			zyl_rafo_vorschub.fb.st_config.b_aktiv := NOT gst_datensatz.st_md.b_wt_transport_simulation;
			zyl_rafo_vorschub.fb(
				st_config:= ,
				bw_nocken_zylinder_einfahren:= ,
				bw_nocken_zylinder_ausfahren:= ,
				uw_nocken_zylinder_einfahren:= ,
				uw_nocken_zylinder_ausfahren:= ,
				b_direkttaste_ausfahren:= ,
				b_direkttaste_mittefahren:= ,
				b_direkttaste_einfahren	:= ,
				e_druckwaechter:= ST_Betriebsfreigaben.e_druckwaechter,
				i16_betriebsart:= gi16_betriebsart,
				b_no_gesteuert_im_norm_betrieb:= ,
				st_ctrl_in:= zyl_rafo_vorschub.st_ctrl.in,
				b_masterachse_hand_dialog_aktiv:= ,
				st_visu:= visu.st_zyl,
				st_ctrl_out=> zyl_rafo_vorschub.st_ctrl.out,
				a_ventil_einfahren=> a_zyl_vorschub_einfahren,
				a_ventil_ausfahren=> a_zyl_vorschub_ausfahren);
	
			zyl_rafo_kamm.fb.st_config.b_aktiv := NOT gst_datensatz.st_md.b_wt_transport_simulation;
			zyl_rafo_kamm.fb(
				st_config:= ,
				bw_nocken_zylinder_einfahren:= ,
				bw_nocken_zylinder_ausfahren:= ,
				uw_nocken_zylinder_einfahren:= ,
				uw_nocken_zylinder_ausfahren:= ,
				b_direkttaste_ausfahren:= ,
				b_direkttaste_mittefahren:= ,
				b_direkttaste_einfahren	:= ,
				e_druckwaechter:= ST_Betriebsfreigaben.e_druckwaechter,
				i16_betriebsart:= gi16_betriebsart,
				b_no_gesteuert_im_norm_betrieb:= ,
				st_ctrl_in:= zyl_rafo_kamm.st_ctrl.in,
				b_masterachse_hand_dialog_aktiv:= ,
				st_visu:= visu.st_zyl,
				st_ctrl_out=> zyl_rafo_kamm.st_ctrl.out,
				a_ventil_einfahren=> ,
				a_ventil_ausfahren=> );
	
			zyl_rafo_vorzentrierer.fb.st_config.b_aktiv := NOT gst_datensatz.st_md.b_wt_transport_simulation;
			zyl_rafo_vorzentrierer.fb(
				st_config:= ,
				bw_nocken_zylinder_einfahren:= ,
				bw_nocken_zylinder_ausfahren:= ,
				uw_nocken_zylinder_einfahren:= ,
				uw_nocken_zylinder_ausfahren:= ,
				b_direkttaste_ausfahren:= ,
				b_direkttaste_mittefahren:= ,
				b_direkttaste_einfahren	:= ,
				e_druckwaechter:= ST_Betriebsfreigaben.e_druckwaechter,
				i16_betriebsart:= gi16_betriebsart,
				b_no_gesteuert_im_norm_betrieb:= ,
				st_ctrl_in:= zyl_rafo_vorzentrierer.st_ctrl.in,
				b_masterachse_hand_dialog_aktiv:= ,
				st_visu:= visu.st_zyl,
				st_ctrl_out=> zyl_rafo_vorzentrierer.st_ctrl.out,
				a_ventil_einfahren=> ,
				a_ventil_ausfahren=> );
	END_CASE
END_IF
END_PROGRAM

(* POU Gemeinsamkeiten17xx/Initialisierung/Startup/ST_Datainit_Zylinder, ST *)
PROGRAM ST_Datainit_Zylinder
VAR
	b_config_fertig			: BOOL := FALSE;
END_VAR
IF	NOT zyl_wt_zentrierer_tisch.fb.st_config.b_config_fertig OR
	NOT zyl_wt_stopper_tisch.fb.st_config.b_config_fertig OR
	NOT zyl_wt_stopper_auslauf.fb.st_config.b_config_fertig OR
	NOT zyl_hublift_rechts_lift.fb.st_config.b_config_fertig OR
	NOT zyl_hublift_rechts_wt_einzug.fb.st_config.b_config_fertig OR
	NOT zyl_hublift_rechts_wt_klinke.fb.st_config.b_config_fertig OR
	NOT zyl_hublift_links_lift.fb.st_config.b_config_fertig OR
	NOT zyl_hublift_links_wt_einzug.fb.st_config.b_config_fertig OR
	NOT zyl_hublift_links_wt_klinke.fb.st_config.b_config_fertig OR
	NOT zyl_hublift_links_stopper.fb.st_config.b_config_fertig OR
	NOT zyl_hublift_links_eingriffschutz.fb.st_config.b_config_fertig OR
	NOT zyl_haspel_li_heben.fb.st_config.b_config_fertig OR
	NOT zyl_haspel_li_abspulen.fb.st_config.b_config_fertig OR
	NOT zyl_haspel_li_sperren.fb.st_config.b_config_fertig OR
	NOT zyl_haspel_re_heben.fb.st_config.b_config_fertig OR
	NOT zyl_haspel_re_abspulen.fb.st_config.b_config_fertig OR
	NOT zyl_haspel_re_sperren.fb.st_config.b_config_fertig OR
	NOT zyl_haspel_verschieben.fb.st_config.b_config_fertig OR
	NOT zyl_bandeinzuege_verschieben.fb.st_config.b_config_fertig OR
	NOT zyl_bawe_vorschub.fb.st_config.b_config_fertig OR
	NOT zyl_bawe_querschub.fb.st_config.b_config_fertig OR
	NOT zyl_bawe_faenger_li.fb.st_config.b_config_fertig OR
	NOT zyl_bawe_faenger_re.fb.st_config.b_config_fertig OR
	NOT zyl_bawe_halter_li.fb.st_config.b_config_fertig OR
	NOT zyl_bawe_halter_re.fb.st_config.b_config_fertig OR
	NOT zyl_wt_stopper_einlauf.fb.st_config.b_config_fertig OR
	NOT zyl_rafo_faenger.fb.st_config.b_config_fertig OR
	NOT zyl_rafo_klemmen.fb.st_config.b_config_fertig OR
	NOT zyl_rafo_vorschub.fb.st_config.b_config_fertig OR
	NOT zyl_rafo_kamm.fb.st_config.b_config_fertig OR
	NOT zyl_rafo_vorzentrierer.fb.st_config.b_config_fertig OR
	NOT zyl_Indexier_Bestueckpos.fb.st_config.b_config_fertig OR
	NOT zyl_Indexier_Einlauf.fb.st_config.b_config_fertig
	THEN

		(* WT Zentrierzylinder am Tisch *)
		zyl_wt_zentrierer_tisch.fb.st_config.b_config_fertig := FALSE;
		zyl_wt_zentrierer_tisch.fb.st_config.b_endlage1_aktiv := FALSE;
		zyl_wt_zentrierer_tisch.fb.st_config.b_endlage2_aktiv := FALSE;
		zyl_wt_zentrierer_tisch.fb.st_config.b_sensor1_aktiv := TRUE;
		zyl_wt_zentrierer_tisch.fb.st_config.b_sensor2_aktiv := TRUE;
		zyl_wt_zentrierer_tisch.fb.st_config.i16_gruppe := 3;
		zyl_wt_zentrierer_tisch.fb.st_config.i16_identnummer := 15;
		zyl_wt_zentrierer_tisch.fb.st_config.i16_meld_startindex := 2280;
		zyl_wt_zentrierer_tisch.fb.st_config.str_beschreibung := ' ';
		zyl_wt_zentrierer_tisch.fb.st_config.str_instanz_name := 'WT Zentrierzylinder am Tisch';
		zyl_wt_zentrierer_tisch.fb.st_config.str_zylinder_typ := '2V4E_EIN_AUS';
		zyl_wt_zentrierer_tisch.fb.st_config.t_ein_aus_fahrzeit := t#0ms;
		zyl_wt_zentrierer_tisch.fb.st_config.t_ueberwachungszeit := t#1000ms;
		zyl_wt_zentrierer_tisch.fb.st_config.i16_tzk_faktor_ausfahren := 100;
		zyl_wt_zentrierer_tisch.fb.st_config.i16_tzk_faktor_einfahren := 100;
		zyl_wt_zentrierer_tisch.fb.st_config.b_config_fertig := TRUE;
		
		(* WT Stoppzylinder am Tisch *)
		zyl_wt_stopper_tisch.fb.st_config.b_config_fertig := FALSE;
		zyl_wt_stopper_tisch.fb.st_config.b_endlage1_aktiv := FALSE;
		zyl_wt_stopper_tisch.fb.st_config.b_endlage2_aktiv := FALSE;
		zyl_wt_stopper_tisch.fb.st_config.b_sensor1_aktiv := TRUE;
		zyl_wt_stopper_tisch.fb.st_config.b_sensor2_aktiv := FALSE;
		zyl_wt_stopper_tisch.fb.st_config.i16_gruppe := 3;
		zyl_wt_stopper_tisch.fb.st_config.i16_identnummer := 16;
		zyl_wt_stopper_tisch.fb.st_config.i16_meld_startindex := 2300;
		zyl_wt_stopper_tisch.fb.st_config.str_beschreibung := ' ';
		zyl_wt_stopper_tisch.fb.st_config.str_instanz_name := 'WT Stoppzylinder am Tisch';

		zyl_wt_stopper_tisch.fb.st_config.t_ein_aus_fahrzeit := t#0ms;
		zyl_wt_stopper_tisch.fb.st_config.t_ueberwachungszeit := t#1000ms;
		zyl_wt_stopper_tisch.fb.st_config.i16_tzk_faktor_ausfahren := 100;
		zyl_wt_stopper_tisch.fb.st_config.i16_tzk_faktor_einfahren := 100;


		IF gst_Datensatz.st_md.b_anwahl_transport_achse THEN
			zyl_wt_stopper_tisch.fb.st_config.str_zylinder_typ := '1V0E_NO';
		ELSE
			zyl_wt_stopper_tisch.fb.st_config.str_zylinder_typ := '2V2E_EIN_AUS';
		END_IF

		zyl_wt_stopper_tisch.fb.st_config.b_config_fertig := TRUE;

		(* WT Stopperzylinder am Auslauf *)
		CASE gst_datensatz.st_md.i16_typ_zelle OF
			KEINE_ZELLE:
				;
			BESTUECKZELLE_1700, RASTERFOLIE:
				zyl_wt_stopper_auslauf.fb.st_config.b_config_fertig := FALSE;
				zyl_wt_stopper_auslauf.fb.st_config.b_endlage1_aktiv := FALSE;
				zyl_wt_stopper_auslauf.fb.st_config.b_endlage2_aktiv := FALSE;
				zyl_wt_stopper_auslauf.fb.st_config.b_sensor1_aktiv := FALSE;
				zyl_wt_stopper_auslauf.fb.st_config.b_sensor2_aktiv := FALSE;
				zyl_wt_stopper_auslauf.fb.st_config.i16_gruppe := 3;
				zyl_wt_stopper_auslauf.fb.st_config.i16_identnummer := 17;
				zyl_wt_stopper_auslauf.fb.st_config.i16_meld_startindex := 2320;
				zyl_wt_stopper_auslauf.fb.st_config.str_beschreibung := ' ';
				zyl_wt_stopper_auslauf.fb.st_config.str_instanz_name := 'WT Stopperzylinder am Auslauf';
				zyl_wt_stopper_auslauf.fb.st_config.str_zylinder_typ := '2V0E';
				zyl_wt_stopper_auslauf.fb.st_config.t_ein_aus_fahrzeit := t#150ms;
				zyl_wt_stopper_auslauf.fb.st_config.t_ueberwachungszeit := t#1000ms;
				zyl_wt_stopper_auslauf.fb.st_config.i16_tzk_faktor_ausfahren := 100;
				zyl_wt_stopper_auslauf.fb.st_config.i16_tzk_faktor_einfahren := 100;
				zyl_wt_stopper_auslauf.fb.st_config.b_config_fertig := TRUE;

			BESTUECKZELLE_1720:
				zyl_wt_stopper_auslauf.fb.st_config.b_config_fertig := FALSE;
				zyl_wt_stopper_auslauf.fb.st_config.b_endlage1_aktiv := FALSE;
				zyl_wt_stopper_auslauf.fb.st_config.b_endlage2_aktiv := FALSE;
				zyl_wt_stopper_auslauf.fb.st_config.b_sensor1_aktiv := FALSE;
				zyl_wt_stopper_auslauf.fb.st_config.b_sensor2_aktiv := FALSE;
				zyl_wt_stopper_auslauf.fb.st_config.i16_gruppe := 3;
				zyl_wt_stopper_auslauf.fb.st_config.i16_identnummer := 17;
				zyl_wt_stopper_auslauf.fb.st_config.i16_meld_startindex := 2320;
				zyl_wt_stopper_auslauf.fb.st_config.str_beschreibung := ' ';
				zyl_wt_stopper_auslauf.fb.st_config.str_instanz_name := 'WT Stopperzylinder am Auslauf';
				zyl_wt_stopper_auslauf.fb.st_config.str_zylinder_typ := '2V2E_EIN_AUS';
				zyl_wt_stopper_auslauf.fb.st_config.t_ein_aus_fahrzeit := t#150ms;
				zyl_wt_stopper_auslauf.fb.st_config.t_ueberwachungszeit := t#1000ms;
				zyl_wt_stopper_auslauf.fb.st_config.i16_tzk_faktor_ausfahren := 100;
				zyl_wt_stopper_auslauf.fb.st_config.i16_tzk_faktor_einfahren := 100;
				zyl_wt_stopper_auslauf.fb.st_config.b_config_fertig := TRUE;
		END_CASE

		(* Hublift-Lift rechts *)
		zyl_hublift_rechts_lift.fb.st_config.b_config_fertig := FALSE;
		zyl_hublift_rechts_lift.fb.st_config.b_endlage1_aktiv := TRUE;
		zyl_hublift_rechts_lift.fb.st_config.b_endlage2_aktiv := FALSE;
		zyl_hublift_rechts_lift.fb.st_config.b_sensor1_aktiv := TRUE;
		zyl_hublift_rechts_lift.fb.st_config.b_sensor2_aktiv := FALSE;
		zyl_hublift_rechts_lift.fb.st_config.i16_gruppe := 4;
		zyl_hublift_rechts_lift.fb.st_config.i16_identnummer := 18;
		zyl_hublift_rechts_lift.fb.st_config.i16_meld_startindex := 2340;
		zyl_hublift_rechts_lift.fb.st_config.str_beschreibung := ' ';
		zyl_hublift_rechts_lift.fb.st_config.str_instanz_name := 'Hublift-Lift rechts';
		zyl_hublift_rechts_lift.fb.st_config.str_zylinder_typ := '2V2E_EIN_AUS';
		zyl_hublift_rechts_lift.fb.st_config.t_ein_aus_fahrzeit := t#0ms;
		zyl_hublift_rechts_lift.fb.st_config.t_ueberwachungszeit := t#3500ms;
		zyl_hublift_rechts_lift.fb.st_config.i16_tzk_faktor_ausfahren := 100;
		zyl_hublift_rechts_lift.fb.st_config.i16_tzk_faktor_einfahren := 100;
		zyl_hublift_rechts_lift.fb.st_config.b_config_fertig := TRUE;
		
		(* Hublift-WT-Einzug rechts *)
		zyl_hublift_rechts_wt_einzug.fb.st_config.b_config_fertig := FALSE;
		zyl_hublift_rechts_wt_einzug.fb.st_config.b_endlage1_aktiv := TRUE;
		zyl_hublift_rechts_wt_einzug.fb.st_config.b_endlage2_aktiv := FALSE;
		zyl_hublift_rechts_wt_einzug.fb.st_config.b_sensor1_aktiv := TRUE;
		zyl_hublift_rechts_wt_einzug.fb.st_config.b_sensor2_aktiv := FALSE;
		zyl_hublift_rechts_wt_einzug.fb.st_config.i16_gruppe := 4;
		zyl_hublift_rechts_wt_einzug.fb.st_config.i16_identnummer := 19;
		zyl_hublift_rechts_wt_einzug.fb.st_config.i16_meld_startindex := 2360;
		zyl_hublift_rechts_wt_einzug.fb.st_config.str_beschreibung := ' ';
		zyl_hublift_rechts_wt_einzug.fb.st_config.str_instanz_name := 'Hublift-WT-Einzug rechts';
		zyl_hublift_rechts_wt_einzug.fb.st_config.str_zylinder_typ := '2V2E_EIN_AUS';
		zyl_hublift_rechts_wt_einzug.fb.st_config.t_ein_aus_fahrzeit := t#0ms;
		zyl_hublift_rechts_wt_einzug.fb.st_config.t_ueberwachungszeit := t#2500ms;
		zyl_hublift_rechts_wt_einzug.fb.st_config.i16_tzk_faktor_ausfahren := 100;
		zyl_hublift_rechts_wt_einzug.fb.st_config.i16_tzk_faktor_einfahren := 100;
		zyl_hublift_rechts_wt_einzug.fb.st_config.b_config_fertig := TRUE;
		
		(* Hublift-WT-Klinke rechts *)
		zyl_hublift_rechts_wt_klinke.fb.st_config.b_config_fertig := FALSE;
		zyl_hublift_rechts_wt_klinke.fb.st_config.b_endlage1_aktiv := TRUE;
		zyl_hublift_rechts_wt_klinke.fb.st_config.b_endlage2_aktiv := FALSE;
		zyl_hublift_rechts_wt_klinke.fb.st_config.b_sensor1_aktiv := TRUE;
		zyl_hublift_rechts_wt_klinke.fb.st_config.b_sensor2_aktiv := FALSE;
		zyl_hublift_rechts_wt_klinke.fb.st_config.i16_gruppe := 4;
		zyl_hublift_rechts_wt_klinke.fb.st_config.i16_identnummer := 20;
		zyl_hublift_rechts_wt_klinke.fb.st_config.i16_meld_startindex := 2380;
		zyl_hublift_rechts_wt_klinke.fb.st_config.str_beschreibung := ' ';
		zyl_hublift_rechts_wt_klinke.fb.st_config.str_instanz_name := 'Hublift-WT-Klinke rechts';
		zyl_hublift_rechts_wt_klinke.fb.st_config.str_zylinder_typ := '2V2E_EIN_AUS';
		zyl_hublift_rechts_wt_klinke.fb.st_config.t_ein_aus_fahrzeit := t#0ms;
		zyl_hublift_rechts_wt_klinke.fb.st_config.t_ueberwachungszeit := t#1500ms;
		zyl_hublift_rechts_wt_klinke.fb.st_config.i16_tzk_faktor_ausfahren := 100;
		zyl_hublift_rechts_wt_klinke.fb.st_config.i16_tzk_faktor_einfahren := 100;
		zyl_hublift_rechts_wt_klinke.fb.st_config.b_config_fertig := TRUE;
		
		(* Hublift-Lift links *)
		zyl_hublift_links_lift.fb.st_config.b_config_fertig := FALSE;
		zyl_hublift_links_lift.fb.st_config.b_endlage1_aktiv := TRUE;
		zyl_hublift_links_lift.fb.st_config.b_endlage2_aktiv := FALSE;
		zyl_hublift_links_lift.fb.st_config.b_sensor1_aktiv := TRUE;
		zyl_hublift_links_lift.fb.st_config.b_sensor2_aktiv := FALSE;
		zyl_hublift_links_lift.fb.st_config.i16_gruppe := 4;
		zyl_hublift_links_lift.fb.st_config.i16_identnummer := 21;
		zyl_hublift_links_lift.fb.st_config.i16_meld_startindex := 2400;
		zyl_hublift_links_lift.fb.st_config.str_beschreibung := ' ';
		zyl_hublift_links_lift.fb.st_config.str_instanz_name := 'Hublift-Lift links';
		zyl_hublift_links_lift.fb.st_config.str_zylinder_typ := '2V2E_EIN_AUS';
		zyl_hublift_links_lift.fb.st_config.t_ein_aus_fahrzeit := t#0ms;
		zyl_hublift_links_lift.fb.st_config.t_ueberwachungszeit := t#3500ms;
		zyl_hublift_links_lift.fb.st_config.i16_tzk_faktor_ausfahren := 100;
		zyl_hublift_links_lift.fb.st_config.i16_tzk_faktor_einfahren := 100;
		zyl_hublift_links_lift.fb.st_config.b_config_fertig := TRUE;
		
		(* Hublift-WT-Einzug links *)
		zyl_hublift_links_wt_einzug.fb.st_config.b_config_fertig := FALSE;
		zyl_hublift_links_wt_einzug.fb.st_config.b_endlage1_aktiv := TRUE;
		zyl_hublift_links_wt_einzug.fb.st_config.b_endlage2_aktiv := FALSE;
		zyl_hublift_links_wt_einzug.fb.st_config.b_sensor1_aktiv := TRUE;
		zyl_hublift_links_wt_einzug.fb.st_config.b_sensor2_aktiv := FALSE;
		zyl_hublift_links_wt_einzug.fb.st_config.i16_gruppe := 4;
		zyl_hublift_links_wt_einzug.fb.st_config.i16_identnummer := 22;
		zyl_hublift_links_wt_einzug.fb.st_config.i16_meld_startindex := 2420;
		zyl_hublift_links_wt_einzug.fb.st_config.str_beschreibung := ' ';
		zyl_hublift_links_wt_einzug.fb.st_config.str_instanz_name := 'Hublift-WT-Einzug links';
		zyl_hublift_links_wt_einzug.fb.st_config.str_zylinder_typ := '2V2E_EIN_AUS';
		zyl_hublift_links_wt_einzug.fb.st_config.t_ein_aus_fahrzeit := t#0ms;
		zyl_hublift_links_wt_einzug.fb.st_config.t_ueberwachungszeit := t#2500ms;
		zyl_hublift_links_wt_einzug.fb.st_config.i16_tzk_faktor_ausfahren := 100;
		zyl_hublift_links_wt_einzug.fb.st_config.i16_tzk_faktor_einfahren := 100;
		zyl_hublift_links_wt_einzug.fb.st_config.b_config_fertig := TRUE;

		(* Hublift-WT-Klinke links *)
		zyl_hublift_links_wt_klinke.fb.st_config.b_config_fertig := FALSE;
		zyl_hublift_links_wt_klinke.fb.st_config.b_endlage1_aktiv := TRUE;
		zyl_hublift_links_wt_klinke.fb.st_config.b_endlage2_aktiv := FALSE;
		zyl_hublift_links_wt_klinke.fb.st_config.b_sensor1_aktiv := TRUE;
		zyl_hublift_links_wt_klinke.fb.st_config.b_sensor2_aktiv := FALSE;
		zyl_hublift_links_wt_klinke.fb.st_config.i16_gruppe := 4;
		zyl_hublift_links_wt_klinke.fb.st_config.i16_identnummer := 23;
		zyl_hublift_links_wt_klinke.fb.st_config.i16_meld_startindex := 2440;
		zyl_hublift_links_wt_klinke.fb.st_config.str_beschreibung := ' ';
		zyl_hublift_links_wt_klinke.fb.st_config.str_instanz_name := 'Hublift-WT-Klinke links';
		zyl_hublift_links_wt_klinke.fb.st_config.str_zylinder_typ := '2V2E_EIN_AUS';
		zyl_hublift_links_wt_klinke.fb.st_config.t_ein_aus_fahrzeit := t#0ms;
		zyl_hublift_links_wt_klinke.fb.st_config.t_ueberwachungszeit := t#1500ms;
		zyl_hublift_links_wt_klinke.fb.st_config.i16_tzk_faktor_ausfahren := 100;
		zyl_hublift_links_wt_klinke.fb.st_config.i16_tzk_faktor_einfahren := 100;
		zyl_hublift_links_wt_klinke.fb.st_config.b_config_fertig := TRUE;

		(* Hublift-Stopper links *)
		zyl_hublift_links_stopper.fb.st_config.b_config_fertig := FALSE;
		zyl_hublift_links_stopper.fb.st_config.b_endlage1_aktiv := TRUE;
		zyl_hublift_links_stopper.fb.st_config.b_endlage2_aktiv := FALSE;
		zyl_hublift_links_stopper.fb.st_config.b_sensor1_aktiv := TRUE;
		zyl_hublift_links_stopper.fb.st_config.b_sensor2_aktiv := FALSE;
		zyl_hublift_links_stopper.fb.st_config.i16_gruppe := 4;
		zyl_hublift_links_stopper.fb.st_config.i16_identnummer := 24;
		zyl_hublift_links_stopper.fb.st_config.i16_meld_startindex := 2460;
		zyl_hublift_links_stopper.fb.st_config.str_beschreibung := ' ';
		zyl_hublift_links_stopper.fb.st_config.str_instanz_name := 'Hublift-Stopper links';
		zyl_hublift_links_stopper.fb.st_config.str_zylinder_typ := '2V2E_EIN_AUS';
		zyl_hublift_links_stopper.fb.st_config.t_ein_aus_fahrzeit := t#0ms;
		zyl_hublift_links_stopper.fb.st_config.t_ueberwachungszeit := t#2000ms;
		zyl_hublift_links_stopper.fb.st_config.i16_tzk_faktor_ausfahren := 100;
		zyl_hublift_links_stopper.fb.st_config.i16_tzk_faktor_einfahren := 100;
		zyl_hublift_links_stopper.fb.st_config.b_config_fertig := TRUE;

		(* zyl_hublift_links_eingriffschutz *)
		zyl_hublift_links_eingriffschutz.fb.st_config.b_config_fertig := FALSE;
		zyl_hublift_links_eingriffschutz.fb.st_config.b_endlage1_aktiv := TRUE;
		zyl_hublift_links_eingriffschutz.fb.st_config.b_endlage2_aktiv := FALSE;
		zyl_hublift_links_eingriffschutz.fb.st_config.b_sensor1_aktiv := TRUE;
		zyl_hublift_links_eingriffschutz.fb.st_config.b_sensor2_aktiv := FALSE;
		zyl_hublift_links_eingriffschutz.fb.st_config.i16_gruppe := 4;
		zyl_hublift_links_eingriffschutz.fb.st_config.i16_identnummer := 44;
		zyl_hublift_links_eingriffschutz.fb.st_config.i16_meld_startindex := 2860;
		zyl_hublift_links_eingriffschutz.fb.st_config.str_beschreibung := ' ';
		zyl_hublift_links_eingriffschutz.fb.st_config.str_instanz_name := 'Hublift links Eingriffschutz';
		zyl_hublift_links_eingriffschutz.fb.st_config.str_zylinder_typ := '2V2E_EIN_AUS';
		zyl_hublift_links_eingriffschutz.fb.st_config.t_ein_aus_fahrzeit := t#0ms;
		zyl_hublift_links_eingriffschutz.fb.st_config.t_ueberwachungszeit := t#4000ms;
		zyl_hublift_links_eingriffschutz.fb.st_config.i16_tzk_faktor_ausfahren := 100;
		zyl_hublift_links_eingriffschutz.fb.st_config.i16_tzk_faktor_einfahren := 100;
		zyl_hublift_links_eingriffschutz.fb.st_config.b_config_fertig := TRUE;
		
		(* Haspel links heben *)
		zyl_haspel_li_heben.fb.st_config.b_config_fertig := FALSE;
		zyl_haspel_li_heben.fb.st_config.b_endlage1_aktiv := FALSE;
		zyl_haspel_li_heben.fb.st_config.b_endlage2_aktiv := FALSE;
		zyl_haspel_li_heben.fb.st_config.b_sensor1_aktiv := FALSE;
		zyl_haspel_li_heben.fb.st_config.b_sensor2_aktiv := FALSE;
		zyl_haspel_li_heben.fb.st_config.i16_gruppe := 2;
		zyl_haspel_li_heben.fb.st_config.i16_identnummer := 7;
		zyl_haspel_li_heben.fb.st_config.i16_meld_startindex := 2120;
		zyl_haspel_li_heben.fb.st_config.str_beschreibung := ' ';
		zyl_haspel_li_heben.fb.st_config.str_instanz_name := 'Haspel links heben';
		zyl_haspel_li_heben.fb.st_config.str_zylinder_typ := '2V1E_AUS';
		zyl_haspel_li_heben.fb.st_config.t_ein_aus_fahrzeit := t#0ms;
		zyl_haspel_li_heben.fb.st_config.t_ueberwachungszeit := t#8s;
		zyl_haspel_li_heben.fb.st_config.i16_tzk_faktor_ausfahren := 100;
		zyl_haspel_li_heben.fb.st_config.i16_tzk_faktor_einfahren := 100;
		zyl_haspel_li_heben.fb.st_config.b_config_fertig := TRUE;
		
		(* Haspel links abspulen *)
		zyl_haspel_li_abspulen.fb.st_config.b_config_fertig := FALSE;
		zyl_haspel_li_abspulen.fb.st_config.b_endlage1_aktiv := FALSE;
		zyl_haspel_li_abspulen.fb.st_config.b_endlage2_aktiv := FALSE;
		zyl_haspel_li_abspulen.fb.st_config.b_sensor1_aktiv := FALSE;
		zyl_haspel_li_abspulen.fb.st_config.b_sensor2_aktiv := FALSE;
		zyl_haspel_li_abspulen.fb.st_config.i16_gruppe := 2;
		zyl_haspel_li_abspulen.fb.st_config.i16_identnummer := 8;
		zyl_haspel_li_abspulen.fb.st_config.i16_meld_startindex := 2140;
		zyl_haspel_li_abspulen.fb.st_config.str_beschreibung := ' ';
		zyl_haspel_li_abspulen.fb.st_config.str_instanz_name := 'Haspel links abspulen';
		zyl_haspel_li_abspulen.fb.st_config.str_zylinder_typ := '2V1E_AUS';
		zyl_haspel_li_abspulen.fb.st_config.t_ein_aus_fahrzeit := t#0ms;
		zyl_haspel_li_abspulen.fb.st_config.t_ueberwachungszeit := t#3s;
		zyl_haspel_li_abspulen.fb.st_config.i16_tzk_faktor_ausfahren := 100;
		zyl_haspel_li_abspulen.fb.st_config.i16_tzk_faktor_einfahren := 100;
		zyl_haspel_li_abspulen.fb.st_config.b_config_fertig := TRUE;
		
		(* Haspel links sperren *)
		zyl_haspel_li_sperren.fb.st_config.b_config_fertig := FALSE;
		zyl_haspel_li_sperren.fb.st_config.b_endlage1_aktiv := FALSE;
		zyl_haspel_li_sperren.fb.st_config.b_endlage2_aktiv := FALSE;
		zyl_haspel_li_sperren.fb.st_config.b_sensor1_aktiv := TRUE;
		zyl_haspel_li_sperren.fb.st_config.b_sensor2_aktiv := FALSE;
		zyl_haspel_li_sperren.fb.st_config.i16_gruppe := 2;
		zyl_haspel_li_sperren.fb.st_config.i16_identnummer := 9;
		zyl_haspel_li_sperren.fb.st_config.i16_meld_startindex := 2160;
		zyl_haspel_li_sperren.fb.st_config.str_beschreibung := ' ';
		zyl_haspel_li_sperren.fb.st_config.str_instanz_name := 'Haspel links sperren';
		zyl_haspel_li_sperren.fb.st_config.str_zylinder_typ := '2V2E_EIN_AUS';
		zyl_haspel_li_sperren.fb.st_config.t_ein_aus_fahrzeit := t#0ms;
		zyl_haspel_li_sperren.fb.st_config.t_ueberwachungszeit := t#1000ms;
		zyl_haspel_li_sperren.fb.st_config.i16_tzk_faktor_ausfahren := 100;
		zyl_haspel_li_sperren.fb.st_config.i16_tzk_faktor_einfahren := 100;
		zyl_haspel_li_sperren.fb.st_config.b_config_fertig := TRUE;
		
		(* Haspel rechts heben *)
		zyl_haspel_re_heben.fb.st_config.b_config_fertig := FALSE;
		zyl_haspel_re_heben.fb.st_config.b_endlage1_aktiv := FALSE;
		zyl_haspel_re_heben.fb.st_config.b_endlage2_aktiv := FALSE;
		zyl_haspel_re_heben.fb.st_config.b_sensor1_aktiv := FALSE;
		zyl_haspel_re_heben.fb.st_config.b_sensor2_aktiv := FALSE;
		zyl_haspel_re_heben.fb.st_config.i16_gruppe := 2;
		zyl_haspel_re_heben.fb.st_config.i16_identnummer := 10;
		zyl_haspel_re_heben.fb.st_config.i16_meld_startindex := 2180;
		zyl_haspel_re_heben.fb.st_config.str_beschreibung := ' ';
		zyl_haspel_re_heben.fb.st_config.str_instanz_name := 'Haspel rechts heben';
		zyl_haspel_re_heben.fb.st_config.str_zylinder_typ := '2V1E_AUS';
		zyl_haspel_re_heben.fb.st_config.t_ein_aus_fahrzeit := t#0ms;
		zyl_haspel_re_heben.fb.st_config.t_ueberwachungszeit := t#8s;
		zyl_haspel_re_heben.fb.st_config.i16_tzk_faktor_ausfahren := 100;
		zyl_haspel_re_heben.fb.st_config.i16_tzk_faktor_einfahren := 100;
		zyl_haspel_re_heben.fb.st_config.b_config_fertig := TRUE;
		
		(* Haspel rechts abspulen *)
		zyl_haspel_re_abspulen.fb.st_config.b_config_fertig := FALSE;
		zyl_haspel_re_abspulen.fb.st_config.b_endlage1_aktiv := FALSE;
		zyl_haspel_re_abspulen.fb.st_config.b_endlage2_aktiv := FALSE;
		zyl_haspel_re_abspulen.fb.st_config.b_sensor1_aktiv := FALSE;
		zyl_haspel_re_abspulen.fb.st_config.b_sensor2_aktiv := FALSE;
		zyl_haspel_re_abspulen.fb.st_config.i16_gruppe := 2;
		zyl_haspel_re_abspulen.fb.st_config.i16_identnummer := 11;
		zyl_haspel_re_abspulen.fb.st_config.i16_meld_startindex := 2200;
		zyl_haspel_re_abspulen.fb.st_config.str_beschreibung := ' ';
		zyl_haspel_re_abspulen.fb.st_config.str_instanz_name := 'Haspel rechts abspulen';
		zyl_haspel_re_abspulen.fb.st_config.str_zylinder_typ := '2V1E_AUS';
		zyl_haspel_re_abspulen.fb.st_config.t_ein_aus_fahrzeit := t#0ms;
		zyl_haspel_re_abspulen.fb.st_config.t_ueberwachungszeit := t#3s;
		zyl_haspel_re_abspulen.fb.st_config.i16_tzk_faktor_ausfahren := 100;
		zyl_haspel_re_abspulen.fb.st_config.i16_tzk_faktor_einfahren := 100;
		zyl_haspel_re_abspulen.fb.st_config.b_config_fertig := TRUE;
		
		(* Haspel rechts sperren *)
		zyl_haspel_re_sperren.fb.st_config.b_config_fertig := FALSE;
		zyl_haspel_re_sperren.fb.st_config.b_endlage1_aktiv := FALSE;
		zyl_haspel_re_sperren.fb.st_config.b_endlage2_aktiv := FALSE;
		zyl_haspel_re_sperren.fb.st_config.b_sensor1_aktiv := FALSE;
		zyl_haspel_re_sperren.fb.st_config.b_sensor2_aktiv := FALSE;
		zyl_haspel_re_sperren.fb.st_config.i16_gruppe := 2;
		zyl_haspel_re_sperren.fb.st_config.i16_identnummer := 12;
		zyl_haspel_re_sperren.fb.st_config.i16_meld_startindex := 2220;
		zyl_haspel_re_sperren.fb.st_config.str_beschreibung := ' ';
		zyl_haspel_re_sperren.fb.st_config.str_instanz_name := 'Haspel rechts sperren';
		zyl_haspel_re_sperren.fb.st_config.str_zylinder_typ := '2V2E_EIN_AUS';
		zyl_haspel_re_sperren.fb.st_config.t_ein_aus_fahrzeit := t#0ms;
		zyl_haspel_re_sperren.fb.st_config.t_ueberwachungszeit := t#1000ms;
		zyl_haspel_re_sperren.fb.st_config.i16_tzk_faktor_ausfahren := 100;
		zyl_haspel_re_sperren.fb.st_config.i16_tzk_faktor_einfahren := 100;
		zyl_haspel_re_sperren.fb.st_config.b_config_fertig := TRUE;
		
		(* Haspel verschieben *)
		zyl_haspel_verschieben.fb.st_config.b_config_fertig := FALSE;
		zyl_haspel_verschieben.fb.st_config.b_endlage1_aktiv := FALSE;
		zyl_haspel_verschieben.fb.st_config.b_endlage2_aktiv := FALSE;
		zyl_haspel_verschieben.fb.st_config.b_sensor1_aktiv := TRUE;
		zyl_haspel_verschieben.fb.st_config.b_sensor2_aktiv := FALSE;
		zyl_haspel_verschieben.fb.st_config.i16_gruppe := 2;
		zyl_haspel_verschieben.fb.st_config.i16_identnummer := 13;
		zyl_haspel_verschieben.fb.st_config.i16_meld_startindex := 2240;
		zyl_haspel_verschieben.fb.st_config.str_beschreibung := ' ';
		zyl_haspel_verschieben.fb.st_config.str_instanz_name := 'Haspel verschieben';
		zyl_haspel_verschieben.fb.st_config.str_zylinder_typ := '2V2E_EIN_AUS';
		zyl_haspel_verschieben.fb.st_config.t_ein_aus_fahrzeit := t#0ms;
		zyl_haspel_verschieben.fb.st_config.t_ueberwachungszeit := t#8s;
		zyl_haspel_verschieben.fb.st_config.i16_tzk_faktor_ausfahren := 100;
		zyl_haspel_verschieben.fb.st_config.i16_tzk_faktor_einfahren := 100;
		zyl_haspel_verschieben.fb.st_config.b_config_fertig := TRUE;
		
		(* Bandeinzüge verschieben *)
		zyl_bandeinzuege_verschieben.fb.st_config.b_config_fertig := FALSE;
		zyl_bandeinzuege_verschieben.fb.st_config.b_endlage1_aktiv := FALSE;
		zyl_bandeinzuege_verschieben.fb.st_config.b_endlage2_aktiv := FALSE;
		zyl_bandeinzuege_verschieben.fb.st_config.b_sensor1_aktiv := TRUE;
		zyl_bandeinzuege_verschieben.fb.st_config.b_sensor2_aktiv := FALSE;
		zyl_bandeinzuege_verschieben.fb.st_config.i16_gruppe := 2;
		zyl_bandeinzuege_verschieben.fb.st_config.i16_identnummer := 14;
		zyl_bandeinzuege_verschieben.fb.st_config.i16_meld_startindex := 2260;
		zyl_bandeinzuege_verschieben.fb.st_config.str_beschreibung := ' ';
		zyl_bandeinzuege_verschieben.fb.st_config.str_instanz_name := 'Bandeinzüge verschieben';
		zyl_bandeinzuege_verschieben.fb.st_config.str_zylinder_typ := '2V2E_EIN_AUS';
		zyl_bandeinzuege_verschieben.fb.st_config.t_ein_aus_fahrzeit := t#0ms;
		zyl_bandeinzuege_verschieben.fb.st_config.t_ueberwachungszeit := t#8000ms;
		zyl_bandeinzuege_verschieben.fb.st_config.i16_tzk_faktor_ausfahren := 100;
		zyl_bandeinzuege_verschieben.fb.st_config.i16_tzk_faktor_einfahren := 100;
		zyl_bandeinzuege_verschieben.fb.st_config.b_config_fertig := TRUE;
		
		(* Bandwechselvorschub *)
		zyl_bawe_vorschub.fb.st_config.b_config_fertig := FALSE;
		zyl_bawe_vorschub.fb.st_config.b_endlage1_aktiv := FALSE;
		zyl_bawe_vorschub.fb.st_config.b_endlage2_aktiv := FALSE;
		zyl_bawe_vorschub.fb.st_config.b_sensor1_aktiv := FALSE;
		zyl_bawe_vorschub.fb.st_config.b_sensor2_aktiv := FALSE;
		zyl_bawe_vorschub.fb.st_config.i16_gruppe := 5;
		zyl_bawe_vorschub.fb.st_config.i16_identnummer := 25;
		zyl_bawe_vorschub.fb.st_config.i16_meld_startindex := 2480;
		zyl_bawe_vorschub.fb.st_config.str_beschreibung := ' ';
		zyl_bawe_vorschub.fb.st_config.str_instanz_name := 'Bandwechselvorschub';
		zyl_bawe_vorschub.fb.st_config.str_zylinder_typ := '2V2E_EIN_AUS';
		zyl_bawe_vorschub.fb.st_config.t_ein_aus_fahrzeit := t#0ms;
		zyl_bawe_vorschub.fb.st_config.t_ueberwachungszeit := t#2000ms;
		zyl_bawe_vorschub.fb.st_config.i16_tzk_faktor_ausfahren := 100;
		zyl_bawe_vorschub.fb.st_config.i16_tzk_faktor_einfahren := 100;
		zyl_bawe_vorschub.fb.st_config.b_config_fertig := TRUE;
		
		(* Bandwechselquerschub *)
		zyl_bawe_querschub.fb.st_config.b_config_fertig := FALSE;
		zyl_bawe_querschub.fb.st_config.b_endlage1_aktiv := FALSE;
		zyl_bawe_querschub.fb.st_config.b_endlage2_aktiv := FALSE;
		zyl_bawe_querschub.fb.st_config.b_sensor1_aktiv := FALSE;
		zyl_bawe_querschub.fb.st_config.b_sensor2_aktiv := FALSE;
		zyl_bawe_querschub.fb.st_config.i16_gruppe := 5;
		zyl_bawe_querschub.fb.st_config.i16_identnummer := 26;
		zyl_bawe_querschub.fb.st_config.i16_meld_startindex := 2500;
		zyl_bawe_querschub.fb.st_config.str_beschreibung := ' ';
		zyl_bawe_querschub.fb.st_config.str_instanz_name := 'Bandwechselquerschub';
		zyl_bawe_querschub.fb.st_config.str_zylinder_typ := '2V2E_EIN_AUS';
		zyl_bawe_querschub.fb.st_config.t_ein_aus_fahrzeit := t#0ms;
		zyl_bawe_querschub.fb.st_config.t_ueberwachungszeit := t#8000ms;
		zyl_bawe_querschub.fb.st_config.i16_tzk_faktor_ausfahren := 100;
		zyl_bawe_querschub.fb.st_config.i16_tzk_faktor_einfahren := 100;
		zyl_bawe_querschub.fb.st_config.b_config_fertig := TRUE;
		
		(* Bandwechselfänger links *)
		zyl_bawe_faenger_li.fb.st_config.b_config_fertig := FALSE;
		zyl_bawe_faenger_li.fb.st_config.b_endlage1_aktiv := FALSE;
		zyl_bawe_faenger_li.fb.st_config.b_endlage2_aktiv := FALSE;
		zyl_bawe_faenger_li.fb.st_config.b_sensor1_aktiv := FALSE;
		zyl_bawe_faenger_li.fb.st_config.b_sensor2_aktiv := FALSE;
		zyl_bawe_faenger_li.fb.st_config.i16_gruppe := 5;
		zyl_bawe_faenger_li.fb.st_config.i16_identnummer := 27;
		zyl_bawe_faenger_li.fb.st_config.i16_meld_startindex := 2520;
		zyl_bawe_faenger_li.fb.st_config.str_beschreibung := ' ';
		zyl_bawe_faenger_li.fb.st_config.str_instanz_name := 'Bandwechselfaenger links';
		zyl_bawe_faenger_li.fb.st_config.str_zylinder_typ := '2V0E';
		zyl_bawe_faenger_li.fb.st_config.t_ein_aus_fahrzeit := t#200ms;
		zyl_bawe_faenger_li.fb.st_config.t_ueberwachungszeit := t#500ms;
		zyl_bawe_faenger_li.fb.st_config.i16_tzk_faktor_ausfahren := 100;
		zyl_bawe_faenger_li.fb.st_config.i16_tzk_faktor_einfahren := 100;
		zyl_bawe_faenger_li.fb.st_config.b_config_fertig := TRUE;
		
		(* Bandwechselfänger rechts *)
		zyl_bawe_faenger_re.fb.st_config.b_config_fertig := FALSE;
		zyl_bawe_faenger_re.fb.st_config.b_endlage1_aktiv := FALSE;
		zyl_bawe_faenger_re.fb.st_config.b_endlage2_aktiv := FALSE;
		zyl_bawe_faenger_re.fb.st_config.b_sensor1_aktiv := FALSE;
		zyl_bawe_faenger_re.fb.st_config.b_sensor2_aktiv := FALSE;
		zyl_bawe_faenger_re.fb.st_config.i16_gruppe := 5;
		zyl_bawe_faenger_re.fb.st_config.i16_identnummer := 28;
		zyl_bawe_faenger_re.fb.st_config.i16_meld_startindex := 2540;
		zyl_bawe_faenger_re.fb.st_config.str_beschreibung := ' ';
		zyl_bawe_faenger_re.fb.st_config.str_instanz_name := 'Bandwechselfaenger rechts';
		zyl_bawe_faenger_re.fb.st_config.str_zylinder_typ := '2V0E';
		zyl_bawe_faenger_re.fb.st_config.t_ein_aus_fahrzeit := t#200ms;
		zyl_bawe_faenger_re.fb.st_config.t_ueberwachungszeit := t#500ms;
		zyl_bawe_faenger_re.fb.st_config.i16_tzk_faktor_ausfahren := 100;
		zyl_bawe_faenger_re.fb.st_config.i16_tzk_faktor_einfahren := 100;
		zyl_bawe_faenger_re.fb.st_config.b_config_fertig := TRUE;
		
		(* Bandwechselhalter links *)
		zyl_bawe_halter_li.fb.st_config.b_config_fertig := FALSE;
		zyl_bawe_halter_li.fb.st_config.b_endlage1_aktiv := FALSE;
		zyl_bawe_halter_li.fb.st_config.b_endlage2_aktiv := FALSE;
		zyl_bawe_halter_li.fb.st_config.b_sensor1_aktiv := FALSE;
		zyl_bawe_halter_li.fb.st_config.b_sensor2_aktiv := FALSE;
		zyl_bawe_halter_li.fb.st_config.i16_gruppe := 5;
		zyl_bawe_halter_li.fb.st_config.i16_identnummer := 29;
		zyl_bawe_halter_li.fb.st_config.i16_meld_startindex := 2560;
		zyl_bawe_halter_li.fb.st_config.str_beschreibung := ' ';
		zyl_bawe_halter_li.fb.st_config.str_instanz_name := 'Bandwechselhalter links';
		zyl_bawe_halter_li.fb.st_config.str_zylinder_typ := '2V0E';
		zyl_bawe_halter_li.fb.st_config.t_ein_aus_fahrzeit := t#200ms;
		zyl_bawe_halter_li.fb.st_config.t_ueberwachungszeit := t#500ms;
		zyl_bawe_halter_li.fb.st_config.i16_tzk_faktor_ausfahren := 100;
		zyl_bawe_halter_li.fb.st_config.i16_tzk_faktor_einfahren := 100;
		zyl_bawe_halter_li.fb.st_config.b_config_fertig := TRUE;
		
		(* Bandwechselhalter rechts *)
		zyl_bawe_halter_re.fb.st_config.b_config_fertig := FALSE;
		zyl_bawe_halter_re.fb.st_config.b_endlage1_aktiv := FALSE;
		zyl_bawe_halter_re.fb.st_config.b_endlage2_aktiv := FALSE;
		zyl_bawe_halter_re.fb.st_config.b_sensor1_aktiv := FALSE;
		zyl_bawe_halter_re.fb.st_config.b_sensor2_aktiv := FALSE;
		zyl_bawe_halter_re.fb.st_config.i16_gruppe := 5;
		zyl_bawe_halter_re.fb.st_config.i16_identnummer := 30;
		zyl_bawe_halter_re.fb.st_config.i16_meld_startindex := 2580;
		zyl_bawe_halter_re.fb.st_config.str_beschreibung := ' ';
		zyl_bawe_halter_re.fb.st_config.str_instanz_name := 'Bandwechselhalter rechts';
		zyl_bawe_halter_re.fb.st_config.str_zylinder_typ := '2V0E';
		zyl_bawe_halter_re.fb.st_config.t_ein_aus_fahrzeit := t#200ms;
		zyl_bawe_halter_re.fb.st_config.t_ueberwachungszeit := t#500ms;
		zyl_bawe_halter_re.fb.st_config.i16_tzk_faktor_ausfahren := 100;
		zyl_bawe_halter_re.fb.st_config.i16_tzk_faktor_einfahren := 100;
		zyl_bawe_halter_re.fb.st_config.b_config_fertig := TRUE;

		(* WT Stopperzylinder am Einlauf *)
		zyl_wt_stopper_einlauf.fb.st_config.b_config_fertig := FALSE;
		zyl_wt_stopper_einlauf.fb.st_config.b_endlage1_aktiv := FALSE;
		zyl_wt_stopper_einlauf.fb.st_config.b_endlage2_aktiv := FALSE;
		zyl_wt_stopper_einlauf.fb.st_config.b_sensor1_aktiv := TRUE;
		zyl_wt_stopper_einlauf.fb.st_config.b_sensor2_aktiv := TRUE;
		zyl_wt_stopper_einlauf.fb.st_config.i16_gruppe := 3;
		zyl_wt_stopper_einlauf.fb.st_config.i16_identnummer := 36;
		zyl_wt_stopper_einlauf.fb.st_config.i16_meld_startindex := 2700;
		zyl_wt_stopper_einlauf.fb.st_config.str_beschreibung := ' ';
		zyl_wt_stopper_einlauf.fb.st_config.str_instanz_name := 'WT Stopperzylinder am Einlauf';
		zyl_wt_stopper_einlauf.fb.st_config.str_zylinder_typ := '1V2E_EIN_AUS';
		zyl_wt_stopper_einlauf.fb.st_config.t_ein_aus_fahrzeit := t#0ms;
		zyl_wt_stopper_einlauf.fb.st_config.t_ueberwachungszeit := t#1000ms;
		zyl_wt_stopper_einlauf.fb.st_config.i16_tzk_faktor_ausfahren := 100;
		zyl_wt_stopper_einlauf.fb.st_config.i16_tzk_faktor_einfahren := 100;
		zyl_wt_stopper_einlauf.fb.st_config.b_config_fertig := TRUE;

		(* Rasterfolien Fänger *)
		zyl_rafo_faenger.fb.st_config.b_config_fertig := FALSE;
		zyl_rafo_faenger.fb.st_config.b_endlage1_aktiv := TRUE;
		zyl_rafo_faenger.fb.st_config.b_endlage2_aktiv := FALSE;
		zyl_rafo_faenger.fb.st_config.b_sensor1_aktiv := TRUE;
		zyl_rafo_faenger.fb.st_config.b_sensor2_aktiv := FALSE;
		zyl_rafo_faenger.fb.st_config.i16_gruppe := 7;
		zyl_rafo_faenger.fb.st_config.i16_identnummer := 37;
		zyl_rafo_faenger.fb.st_config.i16_meld_startindex := 2720;
		zyl_rafo_faenger.fb.st_config.str_beschreibung := ' ';
		zyl_rafo_faenger.fb.st_config.str_instanz_name := 'Rasterfolien Fänger';
		zyl_rafo_faenger.fb.st_config.str_zylinder_typ := '2V1E_AUS';
		zyl_rafo_faenger.fb.st_config.t_ein_aus_fahrzeit := t#100ms;
		zyl_rafo_faenger.fb.st_config.t_ueberwachungszeit := t#500ms;
		zyl_rafo_faenger.fb.st_config.i16_tzk_faktor_ausfahren := 100;
		zyl_rafo_faenger.fb.st_config.i16_tzk_faktor_einfahren := 100;
		zyl_rafo_faenger.fb.st_config.b_config_fertig := TRUE;
		
		(* Rasterfolie Klemmen *)
		zyl_rafo_klemmen.fb.st_config.b_config_fertig := FALSE;
		zyl_rafo_klemmen.fb.st_config.b_endlage1_aktiv := TRUE;
		zyl_rafo_klemmen.fb.st_config.b_endlage2_aktiv := FALSE;
		zyl_rafo_klemmen.fb.st_config.b_sensor1_aktiv := TRUE;
		zyl_rafo_klemmen.fb.st_config.b_sensor2_aktiv := FALSE;
		zyl_rafo_klemmen.fb.st_config.i16_gruppe := 7;
		zyl_rafo_klemmen.fb.st_config.i16_identnummer := 38;
		zyl_rafo_klemmen.fb.st_config.i16_meld_startindex := 2740;
		zyl_rafo_klemmen.fb.st_config.str_beschreibung := ' ';
		zyl_rafo_klemmen.fb.st_config.str_instanz_name := 'Rasterfolie Klemmen';
		zyl_rafo_klemmen.fb.st_config.str_zylinder_typ := '2V1E_AUS';
		zyl_rafo_klemmen.fb.st_config.t_ein_aus_fahrzeit := t#100ms;
		zyl_rafo_klemmen.fb.st_config.t_ueberwachungszeit := t#500ms;
		zyl_rafo_klemmen.fb.st_config.i16_tzk_faktor_ausfahren := 100;
		zyl_rafo_klemmen.fb.st_config.i16_tzk_faktor_einfahren := 100;
		zyl_rafo_klemmen.fb.st_config.b_config_fertig := TRUE;
		
		(* Rasterfolien Vorschub *)
		zyl_rafo_vorschub.fb.st_config.b_config_fertig := FALSE;
		zyl_rafo_vorschub.fb.st_config.b_endlage1_aktiv := TRUE;
		zyl_rafo_vorschub.fb.st_config.b_endlage2_aktiv := FALSE;
		zyl_rafo_vorschub.fb.st_config.b_sensor1_aktiv := TRUE;
		zyl_rafo_vorschub.fb.st_config.b_sensor2_aktiv := FALSE;
		zyl_rafo_vorschub.fb.st_config.i16_gruppe := 7;
		zyl_rafo_vorschub.fb.st_config.i16_identnummer := 39;
		zyl_rafo_vorschub.fb.st_config.i16_meld_startindex := 2760;
		zyl_rafo_vorschub.fb.st_config.str_beschreibung := ' ';
		zyl_rafo_vorschub.fb.st_config.str_instanz_name := 'Rasterplatte Wenden';
		zyl_rafo_vorschub.fb.st_config.str_zylinder_typ := '2V2E_EIN_AUS';
		zyl_rafo_vorschub.fb.st_config.t_ein_aus_fahrzeit := t#100ms;
		zyl_rafo_vorschub.fb.st_config.t_ueberwachungszeit := t#2000ms;
		zyl_rafo_vorschub.fb.st_config.i16_tzk_faktor_ausfahren := 100;
		zyl_rafo_vorschub.fb.st_config.i16_tzk_faktor_einfahren := 100;
		zyl_rafo_vorschub.fb.st_config.b_config_fertig := TRUE;
		
		(* Rasterfolien Kamm *)
		zyl_rafo_kamm.fb.st_config.b_config_fertig := FALSE;
		zyl_rafo_kamm.fb.st_config.b_endlage1_aktiv := TRUE;
		zyl_rafo_kamm.fb.st_config.b_endlage2_aktiv := FALSE;
		zyl_rafo_kamm.fb.st_config.b_sensor1_aktiv := TRUE;
		zyl_rafo_kamm.fb.st_config.b_sensor2_aktiv := FALSE;
		zyl_rafo_kamm.fb.st_config.i16_gruppe := 7;
		zyl_rafo_kamm.fb.st_config.i16_identnummer := 40;
		zyl_rafo_kamm.fb.st_config.i16_meld_startindex := 2780;
		zyl_rafo_kamm.fb.st_config.str_beschreibung := ' ';
		zyl_rafo_kamm.fb.st_config.str_instanz_name := 'Rasterfolien Kamm';
		zyl_rafo_kamm.fb.st_config.str_zylinder_typ := '2V2E_EIN_AUS';
		zyl_rafo_kamm.fb.st_config.t_ein_aus_fahrzeit := t#100ms;
		zyl_rafo_kamm.fb.st_config.t_ueberwachungszeit := t#1500ms;
		zyl_rafo_kamm.fb.st_config.i16_tzk_faktor_ausfahren := 100;
		zyl_rafo_kamm.fb.st_config.i16_tzk_faktor_einfahren := 100;
		zyl_rafo_kamm.fb.st_config.b_config_fertig := TRUE;

		(* Rasterfolien Vorzentrierer *)
		zyl_rafo_vorzentrierer.fb.st_config.b_config_fertig := FALSE;
		zyl_rafo_vorzentrierer.fb.st_config.b_endlage1_aktiv := TRUE;
		zyl_rafo_vorzentrierer.fb.st_config.b_endlage2_aktiv := FALSE;
		zyl_rafo_vorzentrierer.fb.st_config.b_sensor1_aktiv := TRUE;
		zyl_rafo_vorzentrierer.fb.st_config.b_sensor2_aktiv := FALSE;
		zyl_rafo_vorzentrierer.fb.st_config.i16_gruppe := 7;
		zyl_rafo_vorzentrierer.fb.st_config.i16_identnummer := 43;
		zyl_rafo_vorzentrierer.fb.st_config.i16_meld_startindex := 2840;
		zyl_rafo_vorzentrierer.fb.st_config.str_beschreibung := ' ';
		zyl_rafo_vorzentrierer.fb.st_config.str_instanz_name := 'Rasterfolien Vorzentrierer';
		zyl_rafo_vorzentrierer.fb.st_config.str_zylinder_typ := '2V2E_EIN_AUS';
		zyl_rafo_vorzentrierer.fb.st_config.t_ein_aus_fahrzeit := t#100ms;
		zyl_rafo_vorzentrierer.fb.st_config.t_ueberwachungszeit := t#1500ms;
		zyl_rafo_vorzentrierer.fb.st_config.i16_tzk_faktor_ausfahren := 100;
		zyl_rafo_vorzentrierer.fb.st_config.i16_tzk_faktor_einfahren := 100;
		zyl_rafo_vorzentrierer.fb.st_config.b_config_fertig := TRUE;

		(* Indexierzylinder Bestückposition *)
		zyl_Indexier_Bestueckpos.fb.st_config.b_config_fertig := FALSE;
		zyl_Indexier_Bestueckpos.fb.st_config.b_endlage1_aktiv := FALSE;
		zyl_Indexier_Bestueckpos.fb.st_config.b_endlage2_aktiv := FALSE;
		zyl_Indexier_Bestueckpos.fb.st_config.b_sensor1_aktiv := TRUE;
		zyl_Indexier_Bestueckpos.fb.st_config.b_sensor2_aktiv := TRUE;
		zyl_Indexier_Bestueckpos.fb.st_config.i16_gruppe := 3;
		zyl_Indexier_Bestueckpos.fb.st_config.i16_identnummer := 48;
		zyl_Indexier_Bestueckpos.fb.st_config.i16_meld_startindex := 2920;
		zyl_Indexier_Bestueckpos.fb.st_config.str_beschreibung := ' ';
		zyl_Indexier_Bestueckpos.fb.st_config.str_instanz_name := 'Indexierzylinder Bestückposition';
		zyl_Indexier_Bestueckpos.fb.st_config.str_zylinder_typ := '1V2E_EIN_AUS';
		zyl_Indexier_Bestueckpos.fb.st_config.t_ein_aus_fahrzeit := t#0ms;
		zyl_Indexier_Bestueckpos.fb.st_config.t_ueberwachungszeit := t#1000ms;
		zyl_Indexier_Bestueckpos.fb.st_config.i16_tzk_faktor_ausfahren := 100;
		zyl_Indexier_Bestueckpos.fb.st_config.i16_tzk_faktor_einfahren := 100;
		zyl_Indexier_Bestueckpos.fb.st_config.b_config_fertig := TRUE;

		(* Indexierzylinder Einlauf *)
		zyl_Indexier_Einlauf.fb.st_config.b_config_fertig := FALSE;
		zyl_Indexier_Einlauf.fb.st_config.b_endlage1_aktiv := FALSE;
		zyl_Indexier_Einlauf.fb.st_config.b_endlage2_aktiv := FALSE;
		zyl_Indexier_Einlauf.fb.st_config.b_sensor1_aktiv := TRUE;
		zyl_Indexier_Einlauf.fb.st_config.b_sensor2_aktiv := TRUE;
		zyl_Indexier_Einlauf.fb.st_config.i16_gruppe := 3;
		zyl_Indexier_Einlauf.fb.st_config.i16_identnummer := 49;
		zyl_Indexier_Einlauf.fb.st_config.i16_meld_startindex := 2940;
		zyl_Indexier_Einlauf.fb.st_config.str_beschreibung := ' ';
		zyl_Indexier_Einlauf.fb.st_config.str_instanz_name := ' Indexierzylinder Einlauf ';
		zyl_Indexier_Einlauf.fb.st_config.str_zylinder_typ := '1V2E_EIN_AUS';
		zyl_Indexier_Einlauf.fb.st_config.t_ein_aus_fahrzeit := t#0ms;
		zyl_Indexier_Einlauf.fb.st_config.t_ueberwachungszeit := t#1000ms;
		zyl_Indexier_Einlauf.fb.st_config.i16_tzk_faktor_ausfahren := 100;
		zyl_Indexier_Einlauf.fb.st_config.i16_tzk_faktor_einfahren := 100;
		zyl_Indexier_Einlauf.fb.st_config.b_config_fertig := TRUE;
ELSE
	b_config_fertig := FALSE;
END_IF
END_PROGRAM

(* POU EPT Lib/Programmbausteine/ST_start_OSK, ST *)
PROGRAM ST_start_OSK
VAR_INPUT
	bExecute			: BOOL;
END_VAR
VAR
	NT_StartProcess 		:NT_StartProcess;
	b_Start				:BOOL;

	fb_ton_start			:TON;
	fb_r_trig_start			: R_TRIG;

END_VAR
(*Windows Tastatur starten mit der Quttiertaste*)
fb_ton_start(
	IN:=bExecute,
	PT:= t#2s,);

fb_r_trig_start(
	CLK:=fb_ton_start.Q ,
	Q=> b_Start);

NT_StartProcess(
	NETID:='',
	PATHSTR	:='C:\Windows\System32\cmd.exe',
	DIRNAME	:= ,
	COMNDLINE	:='/C C:\WINDOWS\system32\taskkill /f /im osk.exe /t & start /b osk /MAX',
	START		:=b_Start,
	TMOUT		:=T#10s);

IF	NOT NT_StartProcess.BUSY AND b_Start THEN
	b_Start:=FALSE;
END_IF
END_PROGRAM

(* POU Gemeinsamkeiten17xx/Visu/ST_VisuRouter, ST *)
PROGRAM ST_VisuRouter
VAR
END_VAR
(*Anzeige der aktuellen Betriebsart*)
CASE gi16_betriebsart OF
	KEINE:
		visu_hinten.in.betriebsart := visu_hinten.in.texte.txt_variabel[8];

	AUTO:
		visu_hinten.in.betriebsart := visu_hinten.in.texte.txt_variabel[5];

	TIPPEN:
		visu_hinten.in.betriebsart := visu_hinten.in.texte.txt_variabel[6];

	HAND:
		visu_hinten.in.betriebsart := visu_hinten.in.texte.txt_variabel[7];
END_CASE

(*Anzeige des Maschinenstatus*)
CASE gi16_maschinenstatusinfo OF
	KEIN_STATUS:
		visu_hinten.in.s_maschinenstatusinfo := visu_hinten.in.texte.txt_variabel[0];

	STATUS_FEHLER:
		visu_hinten.in.s_maschinenstatusinfo := visu_hinten.in.texte.txt_variabel[1];

	STATUS_FEHLER_QUITTIERT:
		visu_hinten.in.s_maschinenstatusinfo := visu_hinten.in.texte.txt_variabel[2];

	STATUS_BETRIEBSBEREIT:
		visu_hinten.in.s_maschinenstatusinfo := visu_hinten.in.texte.txt_variabel[3];

	STATUS_MASCHINE_ARBEITET:
		visu_hinten.in.s_maschinenstatusinfo := visu_hinten.in.texte.txt_variabel[4];
END_CASE

visu_hinten.in.i16_maschinenstatusinfo := gi16_maschinenstatusinfo;
visu_hinten.in.s_betriebsmeldung := ST_Virtuelle_Masterachse.bm_an_visu_hinten;
visu_hinten.in.i16_position_ist := LREAL_TO_INT(bestueckachse.NcToPlc.ModuloActPos);
visu_hinten.in.i16_typ_zelle := gst_datensatz.st_md.i16_typ_zelle;
visu_hinten.in.i16_typ_bandeinzug:=gst_datensatz.st_wkz.i16_typ_bandeinzug;
visu_hinten.in.band_ID_Puffer_aus:=gst_datensatz.st_md.b_band_ID_Puffer_aus;


visu_hinten.in.texte.txt_zylindernamen[2].s_einfahren:=visu_hinten.in.texte.txt_zylindernamen[0].s_einfahren;
visu_hinten.in.texte.txt_zylindernamen[2].s_ausfahren:=visu_hinten.in.texte.txt_zylindernamen[0].s_ausfahren;
visu_hinten.in.texte.txt_zylindernamen[3].s_einfahren:=visu_hinten.in.texte.txt_zylindernamen[1].s_einfahren;
visu_hinten.in.texte.txt_zylindernamen[3].s_ausfahren:=visu_hinten.in.texte.txt_zylindernamen[1].s_ausfahren;

CASE gst_datensatz.st_md.i16_typ_zelle OF
	KEINE_ZELLE:
		;

	BESTUECKZELLE_1700:

		CASE gst_datensatz.st_wkz.i16_typ_bandeinzug OF
			KEIN_EINZUG:
				;

			STANDARD_2FACH_V2:
				;

			 SERVO:
				(* Die Seitenbezeichnungen (links, rechts) beziehen sich auf die Maschinenvorderseite *)
				(* Haspel Links Heben *)
				zyl_haspel_li_heben.fb.b_direkttaste_ausfahren := visu_hinten.out.zylinder_direkttasten[0].b_ausfahren;
				zyl_haspel_li_heben.fb.b_direkttaste_einfahren := visu_hinten.out.zylinder_direkttasten[0].b_einfahren;
				visu_hinten.in.zylinder_sensoren[0].b_eingefahren := zyl_haspel_li_heben.fb.e_sensor1_eingefahren;
				visu_hinten.in.zylinder_sensoren[0].b_ausgefahren := zyl_haspel_li_heben.fb.e_sensor1_ausgefahren;

				(* Haspel Links Sperren *)
				zyl_haspel_li_sperren.fb.b_direkttaste_ausfahren := visu_hinten.out.zylinder_direkttasten[1].b_ausfahren;
				zyl_haspel_li_sperren.fb.b_direkttaste_einfahren :=  visu_hinten.out.zylinder_direkttasten[1].b_einfahren;
				zyl_haspel_li_abspulen.fb.b_direkttaste_ausfahren:=visu_hinten.out.zylinder_direkttasten[1].b_einfahren; (*Abspulzylinder beim Entriegeln anheben*)
				visu_hinten.in.zylinder_sensoren[1].b_eingefahren := zyl_haspel_li_sperren.fb.e_sensor1_eingefahren;
				visu_hinten.in.zylinder_sensoren[1].b_ausgefahren := zyl_haspel_li_sperren.fb.e_sensor1_ausgefahren;
		
				(* Haspel Rechts Heben *)
				zyl_haspel_re_heben.fb.b_direkttaste_ausfahren := visu_hinten.out.zylinder_direkttasten[2].b_ausfahren;
				zyl_haspel_re_heben.fb.b_direkttaste_einfahren := visu_hinten.out.zylinder_direkttasten[2].b_einfahren;
				visu_hinten.in.zylinder_sensoren[2].b_eingefahren := zyl_haspel_re_heben.fb.e_sensor1_eingefahren;
				visu_hinten.in.zylinder_sensoren[2].b_ausgefahren := zyl_haspel_re_heben.fb.e_sensor1_ausgefahren;
		
				(* Haspel Rechts Sperren *)
				zyl_haspel_re_sperren.fb.b_direkttaste_ausfahren := visu_hinten.out.zylinder_direkttasten[3].b_ausfahren;
				zyl_haspel_re_sperren.fb.b_direkttaste_einfahren := visu_hinten.out.zylinder_direkttasten[3].b_einfahren;
				zyl_haspel_re_abspulen.fb.b_direkttaste_ausfahren:=visu_hinten.out.zylinder_direkttasten[3].b_einfahren; (*Abspulzylinder beim Entriegeln anheben*)
				visu_hinten.in.zylinder_sensoren[3].b_eingefahren := zyl_haspel_re_sperren.fb.e_sensor1_eingefahren;
				visu_hinten.in.zylinder_sensoren[3].b_ausgefahren := zyl_haspel_re_sperren.fb.e_sensor1_ausgefahren;
		
				(* Bandfänger *)
				zyl_bandfaenger.fb.b_direkttaste_ausfahren := visu_hinten.out.zylinder_direkttasten[4].b_ausfahren;
				zyl_bandfaenger.fb.b_direkttaste_einfahren := visu_hinten.out.zylinder_direkttasten[4].b_einfahren;
				visu_hinten.in.zylinder_sensoren[4].b_eingefahren := zyl_bandfaenger.fb.e_sensor1_eingefahren;
				visu_hinten.in.zylinder_sensoren[4].b_ausgefahren := zyl_bandfaenger.fb.e_sensor1_ausgefahren;
		
				(* Bandklemmen *)
				zyl_bandklemmen.fb.b_direkttaste_ausfahren := visu_hinten.out.zylinder_direkttasten[5].b_ausfahren;
				zyl_bandklemmen.fb.b_direkttaste_einfahren := visu_hinten.out.zylinder_direkttasten[5].b_einfahren;
				visu_hinten.in.zylinder_sensoren[5].b_eingefahren := zyl_bandklemmen.fb.e_sensor1_eingefahren;
				visu_hinten.in.zylinder_sensoren[5].b_ausgefahren := zyl_bandklemmen.fb.e_sensor1_ausgefahren;
		
				(* Bandwechselhalter links *)
				zyl_bawe_halter_li.fb.b_direkttaste_ausfahren := visu_hinten.out.zylinder_direkttasten[6].b_ausfahren;
				zyl_bawe_halter_li.fb.b_direkttaste_einfahren := visu_hinten.out.zylinder_direkttasten[6].b_einfahren;
				visu_hinten.in.zylinder_sensoren[6].b_eingefahren := zyl_bawe_halter_li.fb.e_sensor1_eingefahren;
				visu_hinten.in.zylinder_sensoren[6].b_ausgefahren := zyl_bawe_halter_li.fb.e_sensor1_ausgefahren;
		
				(* Bandwechselhalter rechts *)
				zyl_bawe_halter_re.fb.b_direkttaste_ausfahren := visu_hinten.out.zylinder_direkttasten[7].b_ausfahren;
				zyl_bawe_halter_re.fb.b_direkttaste_einfahren := visu_hinten.out.zylinder_direkttasten[7].b_einfahren;
				visu_hinten.in.zylinder_sensoren[7].b_eingefahren := zyl_bawe_halter_re.fb.e_sensor1_eingefahren;
				visu_hinten.in.zylinder_sensoren[7].b_ausgefahren := zyl_bawe_halter_re.fb.e_sensor1_ausgefahren;
		
				(* Bandwechselfänger links *)
				zyl_bawe_faenger_li.fb.b_direkttaste_ausfahren := visu_hinten.out.zylinder_direkttasten[8].b_ausfahren;
				zyl_bawe_faenger_li.fb.b_direkttaste_einfahren := visu_hinten.out.zylinder_direkttasten[8].b_einfahren;
				visu_hinten.in.zylinder_sensoren[8].b_eingefahren := zyl_bawe_faenger_li.fb.e_sensor1_eingefahren;
				visu_hinten.in.zylinder_sensoren[8].b_ausgefahren := zyl_bawe_faenger_li.fb.e_sensor1_ausgefahren;
		
				(* Bandwechselfänger rechts *)
				zyl_bawe_faenger_re.fb.b_direkttaste_ausfahren := visu_hinten.out.zylinder_direkttasten[9].b_ausfahren;
				zyl_bawe_faenger_re.fb.b_direkttaste_einfahren := visu_hinten.out.zylinder_direkttasten[9].b_einfahren;
				visu_hinten.in.zylinder_sensoren[9].b_eingefahren := zyl_bawe_faenger_re.fb.e_sensor1_eingefahren;
				visu_hinten.in.zylinder_sensoren[9].b_ausgefahren := zyl_bawe_faenger_re.fb.e_sensor1_ausgefahren;

				(*Spulenwechsel bie 1700======================*)
				(*Quervorschub*)
				zyl_bawe_querschub.st_ctrl.in.b_ausfahren := visu_hinten.out.zylinder_direkttasten[12].b_ausfahren;
				zyl_bawe_querschub.st_ctrl.in.b_einfahren := visu_hinten.out.zylinder_direkttasten[12].b_einfahren;

				visu_hinten.in.zylinder_sensoren[12].b_eingefahren := zyl_bawe_querschub.fb.e_sensor1_eingefahren;
				visu_hinten.in.zylinder_sensoren[12].b_ausgefahren := zyl_bawe_querschub.fb.e_sensor1_ausgefahren;

				(*Haspel verschieben*)
				zyl_haspel_verschieben.st_ctrl.in.b_ausfahren := visu_hinten.out.zylinder_direkttasten[13].b_ausfahren;
				zyl_haspel_verschieben.st_ctrl.in.b_einfahren := visu_hinten.out.zylinder_direkttasten[13].b_einfahren;

				visu_hinten.in.zylinder_sensoren[13].b_eingefahren := zyl_haspel_verschieben.fb.e_sensor1_eingefahren;
				visu_hinten.in.zylinder_sensoren[13].b_ausgefahren := zyl_haspel_verschieben.fb.e_sensor1_ausgefahren;

				(*Bandeinzug verschieben*)
				zyl_bandeinzuege_verschieben.st_ctrl.in.b_ausfahren := visu_hinten.out.zylinder_direkttasten[14].b_ausfahren;
				zyl_bandeinzuege_verschieben.st_ctrl.in.b_einfahren := visu_hinten.out.zylinder_direkttasten[14].b_einfahren;

				visu_hinten.in.zylinder_sensoren[14].b_eingefahren := zyl_bandeinzuege_verschieben.fb.e_sensor1_eingefahren;
				visu_hinten.in.zylinder_sensoren[14].b_ausgefahren := zyl_bandeinzuege_verschieben.fb.e_sensor1_ausgefahren;

				(* Haspel Links abspulen *)
				zyl_haspel_li_abspulen.fb.b_direkttaste_ausfahren := visu_hinten.out.zylinder_direkttasten[15].b_ausfahren;
				zyl_haspel_li_abspulen.fb.b_direkttaste_einfahren := visu_hinten.out.zylinder_direkttasten[15].b_einfahren;
				visu_hinten.in.zylinder_sensoren[15].b_eingefahren := NOT zyl_haspel_li_abspulen.fb.e_sensor1_ausgefahren;
				visu_hinten.in.zylinder_sensoren[15].b_ausgefahren := zyl_haspel_li_abspulen.fb.e_sensor1_ausgefahren;

				(* Haspel Rechts abspulen *)
				zyl_haspel_re_abspulen.fb.b_direkttaste_ausfahren := visu_hinten.out.zylinder_direkttasten[16].b_ausfahren;
				zyl_haspel_re_abspulen.fb.b_direkttaste_einfahren := visu_hinten.out.zylinder_direkttasten[16].b_einfahren;
				visu_hinten.in.zylinder_sensoren[16].b_eingefahren := NOT zyl_haspel_re_abspulen.fb.e_sensor1_ausgefahren;
				visu_hinten.in.zylinder_sensoren[16].b_ausgefahren := zyl_haspel_re_abspulen.fb.e_sensor1_ausgefahren;


			BANDWECHSLER_V2:(*noch anpassen*)
				(* Die Seitenbezeichnungen (links, rechts) beziehen sich auf die Maschinenvorderseite *)
				(* Haspel Links Heben *)
				zyl_haspel_li_heben.fb.b_direkttaste_ausfahren := visu_hinten.out.zylinder_direkttasten[0].b_ausfahren;
				zyl_haspel_li_heben.fb.b_direkttaste_einfahren := visu_hinten.out.zylinder_direkttasten[0].b_einfahren;
				visu_hinten.in.zylinder_sensoren[0].b_eingefahren := NOT zyl_haspel_li_heben.fb.e_sensor1_ausgefahren;
				visu_hinten.in.zylinder_sensoren[0].b_ausgefahren := zyl_haspel_li_heben.fb.e_sensor1_ausgefahren;

				(* Haspel Links Sperren *)
				zyl_haspel_li_sperren.fb.b_direkttaste_ausfahren := visu_hinten.out.zylinder_direkttasten[1].b_ausfahren;
				zyl_haspel_li_sperren.fb.b_direkttaste_einfahren :=  visu_hinten.out.zylinder_direkttasten[1].b_einfahren;
				zyl_haspel_li_abspulen.fb.b_direkttaste_ausfahren:=visu_hinten.out.zylinder_direkttasten[1].b_einfahren; (*Abspulzylinder beim Entriegeln anheben*)
				visu_hinten.in.zylinder_sensoren[1].b_eingefahren := zyl_haspel_li_sperren.fb.e_sensor1_eingefahren;
				visu_hinten.in.zylinder_sensoren[1].b_ausgefahren := zyl_haspel_li_sperren.fb.e_sensor1_ausgefahren;

				(* Haspel Rechts Heben *)
				zyl_haspel_re_heben.fb.b_direkttaste_ausfahren := visu_hinten.out.zylinder_direkttasten[2].b_ausfahren;
				zyl_haspel_re_heben.fb.b_direkttaste_einfahren := visu_hinten.out.zylinder_direkttasten[2].b_einfahren;
				visu_hinten.in.zylinder_sensoren[2].b_eingefahren := NOT zyl_haspel_re_heben.fb.e_sensor1_ausgefahren;
				visu_hinten.in.zylinder_sensoren[2].b_ausgefahren := zyl_haspel_re_heben.fb.e_sensor1_ausgefahren;

				(* Haspel Rechts Sperren *)
				zyl_haspel_re_sperren.fb.b_direkttaste_ausfahren := visu_hinten.out.zylinder_direkttasten[3].b_ausfahren;
				zyl_haspel_re_sperren.fb.b_direkttaste_einfahren := visu_hinten.out.zylinder_direkttasten[3].b_einfahren;
				zyl_haspel_re_abspulen.fb.b_direkttaste_ausfahren:=visu_hinten.out.zylinder_direkttasten[3].b_einfahren; (*Abspulzylinder beim Entriegeln anheben*)
				visu_hinten.in.zylinder_sensoren[3].b_eingefahren := zyl_haspel_re_sperren.fb.e_sensor1_eingefahren;
				visu_hinten.in.zylinder_sensoren[3].b_ausgefahren := zyl_haspel_re_sperren.fb.e_sensor1_ausgefahren;

				(* Bandfänger *)
				zyl_bandfaenger.fb.b_direkttaste_ausfahren := visu_hinten.out.zylinder_direkttasten[4].b_ausfahren;
				zyl_bandfaenger.fb.b_direkttaste_einfahren := visu_hinten.out.zylinder_direkttasten[4].b_einfahren;
				visu_hinten.in.zylinder_sensoren[4].b_eingefahren := zyl_bandfaenger.fb.a_ventil_einfahren;
				visu_hinten.in.zylinder_sensoren[4].b_ausgefahren := zyl_bandfaenger.fb.a_ventil_ausfahren;
		
				(* Bandklemmen *)
				zyl_bandklemmen.fb.b_direkttaste_ausfahren := visu_hinten.out.zylinder_direkttasten[5].b_ausfahren;
				zyl_bandklemmen.fb.b_direkttaste_einfahren := visu_hinten.out.zylinder_direkttasten[5].b_einfahren;
				visu_hinten.in.zylinder_sensoren[5].b_eingefahren := zyl_bandklemmen.fb.a_ventil_einfahren;
				visu_hinten.in.zylinder_sensoren[5].b_ausgefahren := zyl_bandklemmen.fb.a_ventil_ausfahren;
		
				(* Bandwechselhalter links *)
				zyl_bawe_halter_li.fb.b_direkttaste_ausfahren := visu_hinten.out.zylinder_direkttasten[6].b_ausfahren;
				zyl_bawe_halter_li.fb.b_direkttaste_einfahren := visu_hinten.out.zylinder_direkttasten[6].b_einfahren;
				visu_hinten.in.zylinder_sensoren[6].b_eingefahren := zyl_bawe_halter_li.fb.a_ventil_einfahren;
				visu_hinten.in.zylinder_sensoren[6].b_ausgefahren := zyl_bawe_halter_li.fb.a_ventil_ausfahren;
		
				(* Bandwechselhalter rechts *)
				zyl_bawe_halter_re.fb.b_direkttaste_ausfahren := visu_hinten.out.zylinder_direkttasten[7].b_ausfahren;
				zyl_bawe_halter_re.fb.b_direkttaste_einfahren := visu_hinten.out.zylinder_direkttasten[7].b_einfahren;
				visu_hinten.in.zylinder_sensoren[7].b_eingefahren := zyl_bawe_halter_re.fb.a_ventil_einfahren;
				visu_hinten.in.zylinder_sensoren[7].b_ausgefahren := zyl_bawe_halter_re.fb.a_ventil_ausfahren;
		
				(* Bandwechselfänger links *)
				zyl_bawe_faenger_li.fb.b_direkttaste_ausfahren := visu_hinten.out.zylinder_direkttasten[8].b_ausfahren;
				zyl_bawe_faenger_li.fb.b_direkttaste_einfahren := visu_hinten.out.zylinder_direkttasten[8].b_einfahren;
				visu_hinten.in.zylinder_sensoren[8].b_eingefahren := zyl_bawe_faenger_li.fb.a_ventil_einfahren;
				visu_hinten.in.zylinder_sensoren[8].b_ausgefahren := zyl_bawe_faenger_li.fb.a_ventil_ausfahren;
		
				(* Bandwechselfänger rechts *)
				zyl_bawe_faenger_re.fb.b_direkttaste_ausfahren := visu_hinten.out.zylinder_direkttasten[9].b_ausfahren;
				zyl_bawe_faenger_re.fb.b_direkttaste_einfahren := visu_hinten.out.zylinder_direkttasten[9].b_einfahren;
				visu_hinten.in.zylinder_sensoren[9].b_eingefahren := zyl_bawe_faenger_re.fb.a_ventil_einfahren;
				visu_hinten.in.zylinder_sensoren[9].b_ausgefahren := zyl_bawe_faenger_re.fb.a_ventil_ausfahren;

				(*Spulenwechsel bie 1700======================*)
				(*Quervorschub*)
				zyl_bawe_querschub.st_ctrl.in.b_ausfahren := visu_hinten.out.zylinder_direkttasten[12].b_ausfahren;
				zyl_bawe_querschub.st_ctrl.in.b_einfahren := visu_hinten.out.zylinder_direkttasten[12].b_einfahren;

				visu_hinten.in.zylinder_sensoren[12].b_eingefahren := zyl_bawe_querschub.fb.e_sensor1_eingefahren;
				visu_hinten.in.zylinder_sensoren[12].b_ausgefahren := zyl_bawe_querschub.fb.e_sensor1_ausgefahren;

				(*Haspel verschieben*)
				zyl_haspel_verschieben.st_ctrl.in.b_ausfahren := visu_hinten.out.zylinder_direkttasten[13].b_ausfahren;
				zyl_haspel_verschieben.st_ctrl.in.b_einfahren := visu_hinten.out.zylinder_direkttasten[13].b_einfahren;

				visu_hinten.in.zylinder_sensoren[13].b_eingefahren := zyl_haspel_verschieben.fb.e_sensor1_eingefahren;
				visu_hinten.in.zylinder_sensoren[13].b_ausgefahren := zyl_haspel_verschieben.fb.e_sensor1_ausgefahren;

				(*Bandeinzug verschieben*)
				zyl_bandeinzuege_verschieben.st_ctrl.in.b_ausfahren := visu_hinten.out.zylinder_direkttasten[14].b_ausfahren;
				zyl_bandeinzuege_verschieben.st_ctrl.in.b_einfahren := visu_hinten.out.zylinder_direkttasten[14].b_einfahren;

				visu_hinten.in.zylinder_sensoren[14].b_eingefahren := zyl_bandeinzuege_verschieben.fb.e_sensor1_eingefahren;
				visu_hinten.in.zylinder_sensoren[14].b_ausgefahren := zyl_bandeinzuege_verschieben.fb.e_sensor1_ausgefahren;

				(* Haspel Links abspulen *)
				zyl_haspel_li_abspulen.fb.b_direkttaste_ausfahren := visu_hinten.out.zylinder_direkttasten[15].b_ausfahren;
				zyl_haspel_li_abspulen.fb.b_direkttaste_einfahren := visu_hinten.out.zylinder_direkttasten[15].b_einfahren;
				visu_hinten.in.zylinder_sensoren[15].b_eingefahren := NOT zyl_haspel_li_abspulen.fb.e_sensor1_ausgefahren;
				visu_hinten.in.zylinder_sensoren[15].b_ausgefahren := zyl_haspel_li_abspulen.fb.e_sensor1_ausgefahren;

				(* Haspel Rechts abspulen *)
				zyl_haspel_re_abspulen.fb.b_direkttaste_ausfahren := visu_hinten.out.zylinder_direkttasten[16].b_ausfahren;
				zyl_haspel_re_abspulen.fb.b_direkttaste_einfahren := visu_hinten.out.zylinder_direkttasten[16].b_einfahren;
				visu_hinten.in.zylinder_sensoren[16].b_eingefahren := NOT zyl_haspel_re_abspulen.fb.e_sensor1_ausgefahren;
				visu_hinten.in.zylinder_sensoren[16].b_ausgefahren := zyl_haspel_re_abspulen.fb.e_sensor1_ausgefahren;


		END_CASE

	BESTUECKZELLE_1720:

		CASE gst_datensatz.st_wkz.i16_typ_bandeinzug OF
			KEIN_EINZUG:
				;

			STANDARD_2FACH_V2:(*noch anpassen*)
				(* Die Seitenbezeichnungen (links, rechts) beziehen sich auf die Maschinenvorderseite *)
				(* Haspel Links Heben *)
				zyl_haspel_li_heben.fb.b_direkttaste_ausfahren := visu_hinten.out.zylinder_direkttasten[0].b_ausfahren;
				zyl_haspel_li_heben.fb.b_direkttaste_einfahren := visu_hinten.out.zylinder_direkttasten[0].b_einfahren;
				visu_hinten.in.zylinder_sensoren[0].b_eingefahren := zyl_haspel_li_heben.fb.a_ventil_einfahren;
				visu_hinten.in.zylinder_sensoren[0].b_ausgefahren := zyl_haspel_li_heben.fb.a_ventil_ausfahren;

				(* Haspel Links Sperren *)
				zyl_haspel_li_sperren.fb.b_direkttaste_ausfahren := visu_hinten.out.zylinder_direkttasten[1].b_ausfahren;
				zyl_haspel_li_sperren.fb.b_direkttaste_einfahren :=  visu_hinten.out.zylinder_direkttasten[1].b_einfahren;
				zyl_haspel_li_abspulen.fb.b_direkttaste_ausfahren:=visu_hinten.out.zylinder_direkttasten[1].b_einfahren; (*Abspulzylinder beim Entriegeln anheben*)
				visu_hinten.in.zylinder_sensoren[1].b_eingefahren := zyl_haspel_li_sperren.fb.a_ventil_einfahren;
				visu_hinten.in.zylinder_sensoren[1].b_ausgefahren := zyl_haspel_li_sperren.fb.a_ventil_ausfahren;

				(* Haspel Rechts Heben *)
				zyl_haspel_re_heben.fb.b_direkttaste_ausfahren := visu_hinten.out.zylinder_direkttasten[2].b_ausfahren;
				zyl_haspel_re_heben.fb.b_direkttaste_einfahren := visu_hinten.out.zylinder_direkttasten[2].b_einfahren;
				visu_hinten.in.zylinder_sensoren[2].b_eingefahren := zyl_haspel_re_heben.fb.a_ventil_einfahren;
				visu_hinten.in.zylinder_sensoren[2].b_ausgefahren := zyl_haspel_re_heben.fb.a_ventil_ausfahren;
		
				(* Haspel Rechts Sperren *)
				zyl_haspel_re_sperren.fb.b_direkttaste_ausfahren := visu_hinten.out.zylinder_direkttasten[3].b_ausfahren;
				zyl_haspel_re_sperren.fb.b_direkttaste_einfahren := visu_hinten.out.zylinder_direkttasten[3].b_einfahren;
				zyl_haspel_re_abspulen.fb.b_direkttaste_ausfahren:=visu_hinten.out.zylinder_direkttasten[3].b_einfahren; (*Abspulzylinder beim Entriegeln anheben*)
				visu_hinten.in.zylinder_sensoren[3].b_eingefahren := zyl_haspel_re_sperren.fb.a_ventil_einfahren;
				visu_hinten.in.zylinder_sensoren[3].b_ausgefahren := zyl_haspel_re_sperren.fb.a_ventil_ausfahren;
		
					(* Bandeinzug links: Bandfänger *)
				zyl_bandfaenger_li.fb.b_direkttaste_ausfahren := visu_hinten.out.zylinder_direkttasten[9].b_ausfahren;
				zyl_bandfaenger_li.fb.b_direkttaste_einfahren := visu_hinten.out.zylinder_direkttasten[9].b_einfahren;
				visu_hinten.in.zylinder_sensoren[9].b_eingefahren := zyl_bandfaenger_li.fb.a_ventil_einfahren;
				visu_hinten.in.zylinder_sensoren[9].b_ausgefahren := zyl_bandfaenger_li.fb.a_ventil_ausfahren;

				(* Bandeinzug links: Bandklemmen *)
				zyl_bandklemmen_li.fb.b_direkttaste_ausfahren := visu_hinten.out.zylinder_direkttasten[11].b_ausfahren;
				zyl_bandklemmen_li.fb.b_direkttaste_einfahren := visu_hinten.out.zylinder_direkttasten[11].b_einfahren;
				visu_hinten.in.zylinder_sensoren[11].b_eingefahren := zyl_bandklemmen_li.fb.a_ventil_einfahren;
				visu_hinten.in.zylinder_sensoren[11].b_ausgefahren := zyl_bandklemmen_li.fb.a_ventil_ausfahren;
		
				(* Bandeinzug rechts: Bandfänger *)
				zyl_bandfaenger_re.fb.b_direkttaste_ausfahren := visu_hinten.out.zylinder_direkttasten[8].b_ausfahren;
				zyl_bandfaenger_re.fb.b_direkttaste_einfahren := visu_hinten.out.zylinder_direkttasten[8].b_einfahren;
				visu_hinten.in.zylinder_sensoren[8].b_eingefahren := zyl_bandfaenger_re.fb.a_ventil_einfahren;
				visu_hinten.in.zylinder_sensoren[8].b_ausgefahren := zyl_bandfaenger_re.fb.a_ventil_ausfahren;
		
				(* Bandeinzug rechts: Bandklemmen *)
				zyl_bandklemmen_re.fb.b_direkttaste_ausfahren := visu_hinten.out.zylinder_direkttasten[10].b_ausfahren;
				zyl_bandklemmen_re.fb.b_direkttaste_einfahren := visu_hinten.out.zylinder_direkttasten[10].b_einfahren;
				visu_hinten.in.zylinder_sensoren[10].b_eingefahren := zyl_bandklemmen_re.fb.a_ventil_einfahren;
				visu_hinten.in.zylinder_sensoren[10].b_ausgefahren := zyl_bandklemmen_re.fb.a_ventil_ausfahren;

				(* Bandwechselhalter links *)
				zyl_bawe_halter_li.fb.b_direkttaste_ausfahren := visu_hinten.out.zylinder_direkttasten[7].b_ausfahren;
				zyl_bawe_halter_li.fb.b_direkttaste_einfahren := visu_hinten.out.zylinder_direkttasten[7].b_einfahren;
				visu_hinten.in.zylinder_sensoren[7].b_eingefahren := zyl_bawe_halter_li.fb.e_sensor1_eingefahren;
				visu_hinten.in.zylinder_sensoren[7].b_ausgefahren := zyl_bawe_halter_li.fb.e_sensor1_ausgefahren;
		
				(* Bandwechselhalter rechts *)
				zyl_bawe_halter_re.fb.b_direkttaste_ausfahren := visu_hinten.out.zylinder_direkttasten[6].b_ausfahren;
				zyl_bawe_halter_re.fb.b_direkttaste_einfahren := visu_hinten.out.zylinder_direkttasten[6].b_einfahren;
				visu_hinten.in.zylinder_sensoren[6].b_eingefahren := zyl_bawe_halter_re.fb.e_sensor1_eingefahren;
				visu_hinten.in.zylinder_sensoren[6].b_ausgefahren := zyl_bawe_halter_re.fb.e_sensor1_ausgefahren;

				(* Haspel Links abspulen *)
				zyl_haspel_li_abspulen.fb.b_direkttaste_ausfahren := visu_hinten.out.zylinder_direkttasten[15].b_ausfahren;
				zyl_haspel_li_abspulen.fb.b_direkttaste_einfahren := visu_hinten.out.zylinder_direkttasten[15].b_einfahren;
				visu_hinten.in.zylinder_sensoren[15].b_eingefahren := NOT zyl_haspel_li_abspulen.fb.e_sensor1_ausgefahren;
				visu_hinten.in.zylinder_sensoren[15].b_ausgefahren := zyl_haspel_li_abspulen.fb.e_sensor1_ausgefahren;

				(* Haspel Rechts abspulen *)
				zyl_haspel_re_abspulen.fb.b_direkttaste_ausfahren := visu_hinten.out.zylinder_direkttasten[16].b_ausfahren;
				zyl_haspel_re_abspulen.fb.b_direkttaste_einfahren := visu_hinten.out.zylinder_direkttasten[16].b_einfahren;
				visu_hinten.in.zylinder_sensoren[16].b_eingefahren := NOT zyl_haspel_re_abspulen.fb.e_sensor1_ausgefahren;
				visu_hinten.in.zylinder_sensoren[16].b_ausgefahren := zyl_haspel_re_abspulen.fb.e_sensor1_ausgefahren;

			BANDWECHSLER_V2:
				;

			SERVO:
				;
		END_CASE




	RASTERFOLIE:
		(* Die Seitenbezeichnungen (links, rechts) beziehen sich auf die Maschinenvorderseite *)
		(* Haspel Links Heben *)
		zyl_haspel_li_heben.fb.b_direkttaste_ausfahren := visu_hinten.out.zylinder_direkttasten[0].b_ausfahren;
		zyl_haspel_li_heben.fb.b_direkttaste_einfahren := visu_hinten.out.zylinder_direkttasten[0].b_einfahren;
		visu_hinten.in.zylinder_sensoren[0].b_eingefahren := zyl_haspel_li_heben.fb.e_sensor1_eingefahren;
		visu_hinten.in.zylinder_sensoren[0].b_ausgefahren := zyl_haspel_li_heben.fb.e_sensor1_ausgefahren;

		(* Haspel Links Sperren *)
		zyl_haspel_li_sperren.fb.b_direkttaste_ausfahren := visu_hinten.out.zylinder_direkttasten[1].b_ausfahren;
		zyl_haspel_li_sperren.fb.b_direkttaste_einfahren :=  visu_hinten.out.zylinder_direkttasten[1].b_einfahren;
		zyl_haspel_li_abspulen.fb.b_direkttaste_ausfahren:=visu_hinten.out.zylinder_direkttasten[1].b_einfahren; (*Abspulzylinder beim Entriegeln anheben*)
		visu_hinten.in.zylinder_sensoren[1].b_eingefahren := zyl_haspel_li_sperren.fb.e_sensor1_eingefahren;
		visu_hinten.in.zylinder_sensoren[1].b_ausgefahren := zyl_haspel_li_sperren.fb.e_sensor1_ausgefahren;

		(* Haspel Rechts Heben *)
		zyl_haspel_re_heben.fb.b_direkttaste_ausfahren := visu_hinten.out.zylinder_direkttasten[2].b_ausfahren;
		zyl_haspel_re_heben.fb.b_direkttaste_einfahren := visu_hinten.out.zylinder_direkttasten[2].b_einfahren;
		visu_hinten.in.zylinder_sensoren[2].b_eingefahren := zyl_haspel_re_heben.fb.e_sensor1_eingefahren;
		visu_hinten.in.zylinder_sensoren[2].b_ausgefahren := zyl_haspel_re_heben.fb.e_sensor1_ausgefahren;

		(* Haspel Rechts Sperren *)
		zyl_haspel_re_sperren.fb.b_direkttaste_ausfahren := visu_hinten.out.zylinder_direkttasten[3].b_ausfahren;
		zyl_haspel_re_sperren.fb.b_direkttaste_einfahren := visu_hinten.out.zylinder_direkttasten[3].b_einfahren;
		zyl_haspel_re_abspulen.fb.b_direkttaste_ausfahren:=visu_hinten.out.zylinder_direkttasten[3].b_einfahren; (*Abspulzylinder beim Entriegeln anheben*)
		visu_hinten.in.zylinder_sensoren[3].b_eingefahren := zyl_haspel_re_sperren.fb.e_sensor1_eingefahren;
		visu_hinten.in.zylinder_sensoren[3].b_ausgefahren := zyl_haspel_re_sperren.fb.e_sensor1_ausgefahren;

		(* Folienfänger *)
		zyl_rafo_faenger.fb.b_direkttaste_ausfahren := visu_hinten.out.zylinder_direkttasten[4].b_ausfahren;
		zyl_rafo_faenger.fb.b_direkttaste_einfahren := visu_hinten.out.zylinder_direkttasten[4].b_einfahren;
		visu_hinten.in.zylinder_sensoren[4].b_eingefahren := zyl_rafo_faenger.fb.e_sensor1_eingefahren;
		visu_hinten.in.zylinder_sensoren[4].b_ausgefahren := zyl_rafo_faenger.fb.e_sensor1_ausgefahren;

		(* Folienklemmen *)
		zyl_rafo_klemmen.fb.b_direkttaste_ausfahren := visu_hinten.out.zylinder_direkttasten[5].b_ausfahren;
		zyl_rafo_klemmen.fb.b_direkttaste_einfahren := visu_hinten.out.zylinder_direkttasten[5].b_einfahren;
		visu_hinten.in.zylinder_sensoren[5].b_eingefahren := zyl_rafo_klemmen.fb.e_sensor1_eingefahren;
		visu_hinten.in.zylinder_sensoren[5].b_ausgefahren := zyl_rafo_klemmen.fb.e_sensor1_ausgefahren;
END_CASE
END_PROGRAM

(* POU Gemeinsamkeiten17xx/Allgemeines/ST_Gesamthubzaehler, ST *)
PROGRAM ST_Gesamthubzaehler
VAR
	fb_tp_wz				: TP;
	fb_r_trig				: R_TRIG;
	a_Gesamthubzaehler	 AT %Q* : BOOL;
END_VAR
(* Erzeugung eines zeitkonstanten Zählersignals *)
fb_tp_wz(IN:= nockenschaltwerk_bestueckachse.fb.arr_spur[SP_OT], PT:= t#20ms, Q=> a_Gesamthubzaehler, ET=> );

(* Interner Bestückhubzähler der Maschine*)
fb_r_trig(CLK:= nockenschaltwerk_bestueckachse.fb.arr_spur[SP_OT], Q=> );

IF fb_r_trig.Q THEN
	gst_datensatz.st_md.i32_bestueckhubzaehler := gst_datensatz.st_md.i32_bestueckhubzaehler + 1;
	gst_datensatz.st_md.i32_werkzeughubzaehler := 	gst_datensatz.st_md.i32_werkzeughubzaehler +1;
END_IF

IF gst_datensatz.st_md.i32_bestueckhubzaehler > (EXPT(2,32)) OR gst_datensatz.st_md.i32_bestueckhubzaehler < 0 THEN
	gst_datensatz.st_md.i32_bestueckhubzaehler := 0;
END_IF
END_PROGRAM

(* POU Maschine1700/WT Transport/ST_WT_Transport_Beladen_Achse_1700, ST *)
PROGRAM ST_WT_Transport_Beladen_Achse_1700
VAR_INPUT
	st_config								: struct_config;
	st_ctrl_in								: struct_ctrl_in;
	e_wt_im_aktionsfeld					: BOOL;
END_VAR
VAR_IN_OUT
	st_visu								: struct_visu;
END_VAR
VAR_OUTPUT
	st_ctrl_out							: struct_ctrl_out;
	t_WT_WechselZeit					: TIME := t#0ms;
	t_traegerwechselzeit					: TIME := t#0ms;
	t_Zentrierer_ausfahren					: TIME := t#0ms;
	t_Zentrierer_einfahren					: TIME := t#0ms;
	t_komplett_zyklus						: TIME := t#0ms;
END_VAR
VAR
	fb_ton_uez							: TON;
	fb_ton_wz							: TON;
	fb_ton_quitt							: TON;
	fb_ton_wt_auf_beladepos				: TON;
	fb_tof_wt_auf_beladepos				: TOF;
	fb_r_trig_start							: R_TRIG;
	fb_r_trig_beladepos					: R_TRIG;
	fb_r_trig_beladepos_verlassen			: R_TRIG;
	fb_state_entry							: ST_StateEntry;
	fb_traegerwechselzeit					: ST_Taktzeit;
	fb_WT_WechselZeit					: ST_Taktzeit;
	fb_Zentrierer_ausfahren				: ST_Taktzeit;
	fb_Zentrierer_einfahren					: ST_Taktzeit;
	t_bestueckzeit						: TIME := t#0ms;
	sm_wt_hat_beladepos_nicht_verlassen	: BOOL := FALSE;
	sm_tagnummer_ungueltig				: BOOL := FALSE;
	sm_wt_hat_kein_tag					: BOOL := FALSE;
	sm_tagreader_nicht_fertig				: BOOL := FALSE;
	sm_keine_bandfreigabe				: BOOL := FALSE;
	sm_sensorfehler_beladepos			: BOOL := FALSE;
	bm_abfrage_wt_auf_beladepos			: BOOL := FALSE;
	bm_abfrage_wt_auf_wartepos			: BOOL := FALSE;
	bm_warte_auf_wt_an_stopper			: BOOL := FALSE;
	bMerkerSchrittketteKommtVonInit		: BOOL := FALSE;
	fb_ton_abfrage_wt_auf_beladepos		: TON;
	fb_ton_warte_auf_wt_an_stopper			: TON;
	i									: INT := 0;

	(* zum Testen der Achsen nach Tausch, Bestückbild "Becherspucken", WKZ ausgebaut, Vorschubkontrolle abeschaltet,
	Bit muss von Programmierer geforct werden, zum Beenden Schlüsselschalter auf HAND und Zelle neu starten *)
	b_Dauertest_Achsen					: BOOL := FALSE;

	e_wt_auf_beladepos					AT %I* : BOOL;
	e_wt_beladepos_verlassen				AT %I* : BOOL;
	e_wt_auf_pufferstrecke					AT %I* : BOOL;
END_VAR
(* Zeiten *)
fb_ton_uez(IN:= , PT:= , Q=>  , ET=> );
fb_ton_wz(IN:= , PT:= , Q=> , ET=> );
fb_ton_quitt(IN:= , PT:= t#100ms, Q=> , ET=> );

fb_ton_wt_auf_beladepos(IN:= e_wt_im_aktionsfeld, PT:= t#200ms, Q=> , ET=> );
fb_tof_wt_auf_beladepos(IN:= e_wt_im_aktionsfeld, PT:= t#200ms, Q=> , ET=> );

(* Flanken *)
fb_r_trig_beladepos(CLK:= e_wt_auf_beladepos, Q=> );
fb_r_trig_beladepos_verlassen(CLK:= e_wt_beladepos_verlassen, Q=> );
fb_r_trig_start(CLK:= st_ctrl_in.b_start, Q=> );

(*Trägerwechselzeiten*)
fb_WT_WechselZeit(b_start:= , t_zeit=> );
fb_Zentrierer_ausfahren(b_start:= , t_zeit=> );
fb_Zentrierer_einfahren(b_start:= , t_zeit=> );

(* ==================================Toplevel=================================== *)
IF fb_state_entry.i16_next_step > INIT AND fb_state_entry.i16_next_step < FEHLER THEN
	(* Allgemeine Fehler *)
	IF st_ctrl_in.b_stop THEN
		fb_state_entry.i16_next_step := STOP;
	ELSIF zyl_wt_zentrierer_tisch.st_ctrl.out.b_fehler OR
		zyl_Indexier_Bestueckpos.st_ctrl.out.b_fehler THEN
		fb_state_entry.i16_next_step := FEHLER;
	(* Zylinder im Handbetrieb *)
	ELSIF gi16_betriebsart = HAND AND
		st_visu.st_zyl.i16_nr_zyl_im_handbetrieb = zyl_wt_zentrierer_tisch.fb.st_config.i16_identnummer OR
		st_visu.st_zyl.i16_nr_zyl_im_handbetrieb = zyl_Indexier_Bestueckpos.fb.st_config.i16_identnummer  THEN
		fb_state_entry.i16_next_step := FEHLER;
	END_IF
END_IF

(* ============================Haupt-Schrittkette================================ *)
fb_state_entry(
	i16_next_step:= ,
	i16_pos:= 1,
	s_debugtext:= ,
	E=> ,
	X=> ,
	i16_step=> ,
	i16_last_step=> );

CASE fb_state_entry.i16_step OF
(*=======================================================*)
	INIT_OBJ:
		IF st_config.b_config_fertig THEN
			fb_state_entry.i16_next_step := INIT;
		END_IF

(*=======================================================*)
	INIT:
		IF fb_state_entry.E THEN
			fb_ton_wz.IN := FALSE;
			fb_ton_uez.IN := FALSE;
			fb_ton_quitt.IN := FALSE;
			st_ctrl_out.b_fehler := FALSE;
			st_ctrl_out.b_bereit := FALSE;
			st_ctrl_out.b_fertig := FALSE;
			st_ctrl_out.b_kontroller_start := FALSE;
			zyl_wt_zentrierer_tisch.st_ctrl.in.b_einfahren := FALSE;
			zyl_wt_zentrierer_tisch.st_ctrl.in.b_ausfahren := FALSE;
			zyl_wt_zentrierer_tisch.st_ctrl.in.b_luftlos := FALSE;
			axis_transport_wt_achse.st_ctrl.in.b_start := FALSE;
			axis_z_achse.st_ctrl.in.b_start := FALSE;
			stueckzahlen.st_ctrl.in.b_gutteil_produziert := FALSE;
			sm_wt_hat_beladepos_nicht_verlassen := FALSE;
			sm_tagnummer_ungueltig := FALSE;
			sm_wt_hat_kein_tag := FALSE;
			sm_tagreader_nicht_fertig := FALSE;
			sm_keine_bandfreigabe := FALSE;
			bm_abfrage_wt_auf_beladepos := FALSE;
			bm_warte_auf_wt_an_stopper := FALSE;
			balluff_tag_reader.st_ctrl.in.b_start_lesen := FALSE;
			balluff_tag_reader.st_ctrl.in.b_start_schreiben := FALSE;
			zyl_Indexier_Bestueckpos.st_ctrl.in.b_ausfahren := FALSE;
			zyl_Indexier_Bestueckpos.st_ctrl.in.b_einfahren := FALSE;
			bMerkerSchrittketteKommtVonInit := TRUE;
		END_IF

		(*-----------------------Weiterschaltbedingungen----------------------------*)
		IF st_ctrl_in.b_init THEN
			zyl_wt_zentrierer_tisch.st_ctrl.in.b_quittieren := FALSE;
			zyl_Indexier_Bestueckpos.st_ctrl.in.b_quittieren := FALSE;
			fb_state_entry.i16_next_step := 20;
		END_IF

(*=======================================================*)
	20: fb_state_entry.s_debugtext := 'Initialisierung: Stopper an Bestücktisch ausfahren und Zentrierer einfahren';

		(*-----------------------Weiterschaltbedingungen----------------------------*)
		IF e_wt_im_aktionsfeld THEN
			fb_state_entry.i16_next_step := 25;
		ELSE
			fb_state_entry.i16_next_step := 22;
		END_IF

(*=======================================================*)
	22: fb_state_entry.s_debugtext := 'Initialisierung: Stopper an Bestücktisch ausfahren und Zentrierer einfahren';

		IF fb_state_entry.E THEN
			zyl_wt_zentrierer_tisch.st_ctrl.in.b_einfahren := TRUE;
		END_IF

		(*-----------------------Weiterschaltbedingungen----------------------------*)
		IF  zyl_wt_zentrierer_tisch.st_ctrl.out.b_eingefahren THEN
			zyl_wt_zentrierer_tisch.st_ctrl.in.b_einfahren := FALSE;
			fb_state_entry.i16_next_step := 30;
		END_IF

(*=======================================================*)
	25: fb_state_entry.s_debugtext := 'Initialisierung: Stopper an Bestücktisch ausfahren und Zentrierer einfahren';

		IF fb_state_entry.E THEN
			zyl_wt_zentrierer_tisch.st_ctrl.in.b_ausfahren := TRUE;
		END_IF

		(*-----------------------Weiterschaltbedingungen----------------------------*)
		IF  zyl_wt_zentrierer_tisch.st_ctrl.out.b_ausgefahren THEN
			zyl_wt_zentrierer_tisch.st_ctrl.in.b_ausfahren := FALSE;
			fb_state_entry.i16_next_step := 30;
		END_IF

(*=======================================================*)
	30: fb_state_entry.s_debugtext := 'Indexierzylinder wieder einfahren';

		IF fb_state_entry.E THEN
			zyl_Indexier_Bestueckpos.st_ctrl.in.b_ausfahren:= TRUE;
		END_IF

		(*-----------------------Weiterschaltbedingungen----------------------------*)
		IF zyl_Indexier_Bestueckpos.st_ctrl.out.b_ausgefahren THEN
			zyl_Indexier_Bestueckpos.st_ctrl.in.b_ausfahren:= FALSE;
			fb_state_entry.i16_next_step := 35;
		END_IF

(*=======================================================*)
	35: fb_state_entry.s_debugtext := 'warten auf Achse bereit';

		(*-----------------------Weiterschaltbedingungen----------------------------*)
		IF	axis_transport_wt_achse.st_ctrl.out.b_bereit AND
			NOT axis_transport_wt_achse.st_ctrl.in.b_start THEN
			fb_state_entry.i16_next_step := 40;
		END_IF

(*=======================================================*)
	40: fb_state_entry.s_debugtext := 'Fahre Achse wieder zurück';

		IF fb_state_entry.E THEN
			ST_WT_Transport_Achse.lr_Achspos_in:=gst_datensatz.st_md.st_md_transport_wt_achse.lr_startposition;
			ST_WT_Transport_Achse.lr_Velo_in:= gst_datensatz.st_md.r_geschwindigkeit_achse_transport;
			ST_WT_Transport_Achse.enu_cmd_in:=MOVE_ABSOLUTE;
			axis_transport_wt_achse.st_ctrl.in.b_start := TRUE;
		END_IF

		(*-----------------------Weiterschaltbedingungen----------------------------*)
		IF  axis_transport_wt_achse.st_ctrl.out.b_busy THEN
			axis_transport_wt_achse.st_ctrl.in.b_start := FALSE;
			fb_state_entry.i16_next_step := 50;
		END_IF

(*=======================================================*)
	50: fb_state_entry.s_debugtext := 'warten auf Achse hinten fertig';

		(*-----------------------Weiterschaltbedingungen----------------------------*)
		IF	axis_transport_wt_achse.st_ctrl.out.b_fertig  THEN
			fb_state_entry.i16_next_step := BEREIT;
		END_IF

(*=======================================================*)
	BEREIT:	fb_state_entry.s_debugtext := 'Warte auf Start von Kontroller';

		IF fb_state_entry.E THEN
			st_ctrl_out.b_bereit := TRUE;
			st_ctrl_out.b_fertig := TRUE;
			stueckzahlen.st_ctrl.in.b_gutteil_produziert := FALSE;
		END_IF

		(*-----------------------Weiterschaltbedingungen----------------------------*)
		IF st_config.b_station_aktiv OR st_config.b_station_in_simulation THEN

		(* WT Transport aktiv oder in Simulation *)
			IF 	st_ctrl_in.b_start  AND
				((NOT ST_Virtuelle_Masterachse.b_merker_bandende_links  AND
 				NOT ST_Virtuelle_Masterachse.b_merker_bandende_rechts) OR
				gst_datensatz.st_md.b_auto_Bandwechsel) THEN
			(* WT Transport gestartet *)
				st_ctrl_out.b_fertig := FALSE;
				fb_ton_wz.IN := FALSE;
				st_ctrl_out.b_kontroller_start := TRUE;
				(* Abfrage, ob Schrittkette von Init kommt und ob WT auf Beladepos ist *)
				IF bMerkerSchrittketteKommtVonInit AND
					e_wt_auf_beladepos THEN
					fb_state_entry.i16_next_step := 150;	(* WT auslesen und prüfen, ob dieser schon bestückt wurde *)
				ELSE
					fb_state_entry.i16_next_step := 110;
				END_IF
			END_IF

		(* WT-Transport nicht aktiv  *)
		ELSE
			IF fb_r_trig_start.Q THEN
				(* Nur Z-Achse gestartet *)
				st_ctrl_out.b_fertig := FALSE;
				fb_ton_wz.IN := FALSE;
				fb_state_entry.i16_next_step := 500;
			END_IF
		END_IF

		IF fb_state_entry.X THEN
			bMerkerSchrittketteKommtVonInit := FALSE;
		END_IF

(*=======================================================*)
	110: fb_state_entry.s_debugtext := 'WT-Abfrage auf Beladeposition';

		IF fb_state_entry.E THEN
			bm_abfrage_wt_auf_beladepos := TRUE;
		END_IF

		(*-----------------------Weiterschaltbedingungen----------------------------*)
		IF e_wt_im_aktionsfeld THEN
			(* Ein WT ist anwesend zum rausschicken *)
			IF NOT ST_WT_Transport_Abgabe.e_wt_auf_abgabepos THEN
				(* Erst wenn kein Stau vorhanden ist, dann wird der WT weiter gelassen *)
				fb_state_entry.i16_next_step := 115;
			END_IF
		ELSE	(* Kein WT da, deshalb einen holen *)
			fb_state_entry.i16_next_step := 130;
		END_IF

		IF fb_state_entry.X THEN
			bm_abfrage_wt_auf_beladepos := FALSE;
			st_ctrl_out.b_kontroller_start := FALSE;
		END_IF

(*=======================================================*)
	115: fb_state_entry.s_debugtext := 'Indexierzylinder Bestückposition ausfahren (WT festhalten)';

		IF fb_state_entry.E THEN
			zyl_Indexier_Bestueckpos.st_ctrl.in.b_einfahren:= TRUE;
		END_IF

		(*-----------------------Weiterschaltbedingungen----------------------------*)
		IF zyl_Indexier_Bestueckpos.st_ctrl.out.b_eingefahren THEN
			zyl_Indexier_Bestueckpos.st_ctrl.in.b_einfahren:= FALSE;
			fb_state_entry.i16_next_step := 120;
		END_IF

(*=======================================================*)
	120: fb_state_entry.s_debugtext := 'WT-Zentrierer einfahren';

		IF fb_state_entry.E THEN
			zyl_wt_zentrierer_tisch.st_ctrl.in.b_einfahren := TRUE;
			fb_Zentrierer_einfahren(b_start:= TRUE, t_zeit=> );
		END_IF

		(*-----------------------Weiterschaltbedingungen----------------------------*)
		IF zyl_wt_zentrierer_tisch.st_ctrl.out.b_eingefahren THEN
			zyl_wt_zentrierer_tisch.st_ctrl.in.b_einfahren := FALSE;
			fb_Zentrierer_einfahren(b_start:= FALSE, t_zeit=>t_Zentrierer_einfahren);
			fb_state_entry.i16_next_step := 130;
		END_IF

(*=======================================================*)
	130: fb_state_entry.s_debugtext := 'WT ist auf Warteposition und mit Indexierzylinder fixiert, wenn 2 Sekunden kein WT aus der vorherigen Zelle kommt wird der WT weitergeschickt';

		IF fb_state_entry.E THEN
			bm_abfrage_wt_auf_wartepos := TRUE;
		END_IF

		(*-----------------------Weiterschaltbedingungen----------------------------*)
		IF ST_WT_Transport_Warteposition_1700.e_wt_auf_wartepos_1700 AND
			 zyl_Indexier_Einlauf.st_ctrl.out.b_eingefahren AND
			ST_WT_Transport_Warteposition_1700.b_helpStartAchse AND
			zyl_wt_stopper_tisch.st_ctrl.out.b_eingefahren THEN
			fb_state_entry.i16_next_step := 135;
		ELSIF fb_state_entry.fb_ton_Step.ET >= T#2S AND
			 zyl_Indexier_Bestueckpos.st_ctrl.out.b_eingefahren THEN
			fb_state_entry.i16_next_step := 132;
		END_IF

(*=======================================================*)
	132: fb_state_entry.s_debugtext := 'Warten bis kein WT mehr auf der Abgabeposition steht';

		(*-----------------------Weiterschaltbedingungen----------------------------*)
		IF NOT ST_WT_Transport_Abgabe.e_wt_auf_abgabepos THEN
			fb_state_entry.i16_next_step := 135;
		END_IF

(*=======================================================*)
	135: fb_state_entry.s_debugtext := 'warten auf Achse bereit';

		(*-----------------------Weiterschaltbedingungen----------------------------*)
		IF	axis_transport_wt_achse.st_ctrl.out.b_bereit AND
			NOT axis_transport_wt_achse.st_ctrl.out.b_busy  AND
			NOT axis_transport_wt_achse.st_ctrl.in.b_start AND
			((ST_WT_Transport_Warteposition_1700.b_helpStartAchse AND
			ST_WT_Transport_Warteposition_1700.e_wt_auf_wartepos_1700)
			OR
			(zyl_Indexier_Einlauf.st_ctrl.out.b_ausgefahren AND
			NOT ST_WT_Transport_Warteposition_1700.e_wt_auf_wartepos_1700))  THEN
			fb_state_entry.i16_next_step := 140;
		END_IF

(*=======================================================*)
	140: fb_state_entry.s_debugtext := 'Fahre Achse nach vorne -> Bestückposition';

		IF fb_state_entry.E THEN
			ST_WT_Transport_Achse.lr_Achspos_in:=gst_datensatz.st_md.st_md_transport_wt_achse.lr_wt_uebergabepos;
			ST_WT_Transport_Achse.lr_Velo_in:= gst_datensatz.st_md.r_geschwindigkeit_achse_transport;
			ST_WT_Transport_Achse.enu_cmd_in:=MOVE_ABSOLUTE;
			axis_transport_wt_achse.st_ctrl.in.b_start := TRUE;

			st_ctrl_out.b_kontroller_start := TRUE;
		END_IF

		(*-----------------------Weiterschaltbedingungen----------------------------*)
		IF	axis_transport_wt_achse.st_ctrl.out.b_busy THEN
			axis_transport_wt_achse.st_ctrl.in.b_start := FALSE;
			fb_state_entry.i16_next_step := 145;
		END_IF

(*=======================================================*)
	145: fb_state_entry.s_debugtext := 'warten auf Achse vorne fertig';

		(*-----------------------Weiterschaltbedingungen----------------------------*)
		IF	axis_transport_wt_achse.st_ctrl.out.b_fertig THEN
			IF  zyl_Indexier_Einlauf.st_ctrl.out.b_eingefahren THEN
				fb_state_entry.i16_next_step := 147;	(* Neuer WT kommt von Warteposition *)
			ELSE
				fb_state_entry.i16_next_step := 300;	(* Es kommt kein neuer WT *)
			END_IF
		END_IF

		IF fb_state_entry.X THEN
			st_ctrl_out.b_kontroller_start := FALSE;
		END_IF

(*=======================================================*)
	147: fb_state_entry.s_debugtext := 'Prüfe, ob WT auf Beladeposition angekommen ist';

		(*-----------------------Weiterschaltbedingungen----------------------------*)
		IF e_wt_im_aktionsfeld AND
			NOT  ST_WT_Transport_Warteposition_1700.e_wt_auf_wartepos_1700  THEN
			fb_state_entry.i16_next_step := 150;
		ELSE
			sm_wt_hat_beladepos_nicht_verlassen := TRUE;
			fb_state_entry.i16_next_step := FEHLER;
		END_IF

(*=======================================================*)
	150: (*erst weiter wenn Abgabe funktioniert hat  *)

		IF 	NOT ST_WT_Transport_Abgabe.sm_wt_hat_abgabepos_nicht_verlassen THEN
			fb_state_entry.i16_next_step := 152;
		END_IF

		IF fb_state_entry.fb_ton_Step.ET > t#5s  THEN
			fb_state_entry.i16_next_step := STOP;
		END_IF

(*=======================================================*)
	152: (* WT-Zentrierer ausfahren *)

		IF fb_state_entry.E THEN
			zyl_wt_zentrierer_tisch.st_ctrl.in.b_ausfahren := TRUE;
			zyl_Indexier_Bestueckpos.st_ctrl.in.b_ausfahren:= TRUE;
			fb_Zentrierer_ausfahren(b_start:= TRUE, t_zeit=> );
		END_IF

		(*-----------------------Weiterschaltbedingungen----------------------------*)
		IF zyl_wt_zentrierer_tisch.st_ctrl.out.b_ausgefahren AND
			NOT ST_TippTasten.b_einfaedeln_aktiv AND
			NOT ST_Virtuelle_Masterachse.b_merker_bandende_links  AND
 			NOT ST_Virtuelle_Masterachse.b_merker_bandende_rechts AND
			zyl_Indexier_Bestueckpos.st_ctrl.out.b_ausgefahren THEN
			fb_Zentrierer_ausfahren(b_start:= FALSE, t_zeit=> t_Zentrierer_ausfahren);
			zyl_wt_zentrierer_tisch.st_ctrl.in.b_ausfahren := FALSE;
			fb_state_entry.i16_next_step := 155;
		END_IF

(*=======================================================*)
	155: fb_state_entry.s_debugtext := 'WT-Tag mit RFID-Lesegerät abfragen';

		(*-----------------------Weiterschaltbedingungen----------------------------*)
		IF  fb_state_entry.fb_ton_Step.ET >= T#100MS THEN
			IF e_wt_im_aktionsfeld THEN
				(* Tag auslesen *)
				fb_state_entry.i16_next_step := 160;
			ELSE
				(* Kein Tag auf WT *)
				sm_wt_hat_kein_tag := TRUE;
				fb_state_entry.i16_next_step := FEHLER;
			END_IF
		END_IF

(*=======================================================*)
	160: fb_state_entry.s_debugtext := 'Prüfe ob Simulation';

		(*-----------------------Weiterschaltbedingungen----------------------------*)
		IF 	st_config.b_station_in_simulation AND
			NOT visu.b_inbetriebnahme THEN
			fb_state_entry.i16_next_step := 300;
		ELSE
			fb_state_entry.i16_next_step := 170;
		END_IF

(*=======================================================*)
	170: fb_state_entry.s_debugtext := 'Z-Achse und anschliessend Bestückachse wird gestartet';

		IF fb_state_entry.E THEN
			axis_z_achse.st_ctrl.in.b_start := TRUE;
			(*Zeitmessung Trägerwechsel stoppen und ausgeben*)
			fb_WT_WechselZeit(b_start:=FALSE , t_zeit=>t_WT_WechselZeit );
		END_IF

		(*-----------------------Weiterschaltbedingungen----------------------------*)
		IF axis_z_achse.st_ctrl.out.b_busy THEN
			axis_z_achse.st_ctrl.in.b_start := FALSE;
			fb_state_entry.i16_next_step := 175;
		END_IF

(*=======================================================*)
	175: (*erst weiter wenn Abgabe funktioniert hat  *)

		IF 	NOT ST_WT_Transport_Abgabe.sm_wt_hat_abgabepos_nicht_verlassen THEN
			fb_state_entry.i16_next_step := 180;
		END_IF

		IF fb_state_entry.fb_ton_Step.ET > t#5s  THEN
			fb_state_entry.i16_next_step := STOP;
		END_IF

(*=======================================================*)
	180: fb_state_entry.s_debugtext := 'Indexierzylinder wieder einfahren (WT freigeben)';

		IF fb_state_entry.E THEN
			zyl_Indexier_Bestueckpos.st_ctrl.in.b_ausfahren:= TRUE;
		END_IF

		(*-----------------------Weiterschaltbedingungen----------------------------*)
		IF zyl_Indexier_Bestueckpos.st_ctrl.out.b_ausgefahren AND
			zyl_Indexier_Einlauf.st_ctrl.out.b_ausgefahren THEN
			zyl_Indexier_Bestueckpos.st_ctrl.in.b_ausfahren:= FALSE;
			fb_state_entry.i16_next_step := 190;
		END_IF

(*=======================================================*)
	190: fb_state_entry.s_debugtext := 'warten auf Achse bereit';

		(*-----------------------Weiterschaltbedingungen----------------------------*)
		IF	axis_transport_wt_achse.st_ctrl.out.b_bereit AND
			NOT axis_transport_wt_achse.st_ctrl.out.b_busy  AND
			NOT axis_transport_wt_achse.st_ctrl.in.b_start THEN
			fb_state_entry.i16_next_step := 200;
		END_IF

(*=======================================================*)
	200: fb_state_entry.s_debugtext := 'Fahre Achse wieder zurück';

		IF fb_state_entry.E THEN
			ST_WT_Transport_Achse.lr_Achspos_in:=gst_datensatz.st_md.st_md_transport_wt_achse.lr_startposition;
			ST_WT_Transport_Achse.lr_Velo_in:= gst_datensatz.st_md.r_geschwindigkeit_achse_transport;
			ST_WT_Transport_Achse.enu_cmd_in:=MOVE_ABSOLUTE;
			axis_transport_wt_achse.st_ctrl.in.b_start := TRUE;
		END_IF

		(*-----------------------Weiterschaltbedingungen----------------------------*)
		IF	axis_transport_wt_achse.st_ctrl.out.b_busy  THEN
			axis_transport_wt_achse.st_ctrl.in.b_start := FALSE;
			fb_state_entry.i16_next_step := 210;
		END_IF

(*=======================================================*)
	210: fb_state_entry.s_debugtext := 'warten auf Achse hinten fertig';

		(*-----------------------Weiterschaltbedingungen----------------------------*)
		IF	axis_transport_wt_achse.st_ctrl.out.b_fertig  THEN
			fb_state_entry.i16_next_step := 220;
		END_IF

(*=======================================================*)
	220: fb_state_entry.s_debugtext := 'Indexierzylinder Bestückposition ausfahren (WT festhalten)';

		IF fb_state_entry.E THEN
			zyl_Indexier_Bestueckpos.st_ctrl.in.b_einfahren:= TRUE;
		END_IF

		(*-----------------------Weiterschaltbedingungen----------------------------*)
		IF zyl_Indexier_Bestueckpos.st_ctrl.out.b_eingefahren THEN
			zyl_Indexier_Bestueckpos.st_ctrl.in.b_einfahren:= FALSE;
			fb_state_entry.i16_next_step := 230;
		END_IF

(*=======================================================*)
	230: fb_state_entry.s_debugtext := 'Bestückachse ist fertig';

		(*-----------------------Weiterschaltbedingungen----------------------------*)
		IF axis_virt_master.st_ctrl.out.b_fertig THEN
			IF axis_z_achse.st_ctrl.out.b_fertig THEN
				(*Zeitmessung Trägerwechsel starten*)
				fb_WT_WechselZeit(b_start:=TRUE , t_zeit=> );
				(*Zeitmessung zusammenfassen*)
				t_bestueckzeit:=ST_Z_Achse.t_Bestueckung;
				t_traegerwechselzeit:=t_WT_WechselZeit + ST_Z_Achse.t_Z_Achse_einfahren + ST_Z_Achse.t_Z_Achse_ausfahren;
				t_komplett_zyklus:= t_traegerwechselzeit + t_bestueckzeit;

				stueckzahlen.st_ctrl.in.b_gutteil_produziert := TRUE;

				st_ctrl_out.b_kontroller_start := FALSE;
				fb_state_entry.i16_next_step := BEREIT;
			END_IF
		END_IF

(*=======================================================*)
	300: fb_state_entry.s_debugtext := 'Indexierzylinder wieder einfahren (WT freigeben)';

		IF fb_state_entry.E THEN
			zyl_Indexier_Bestueckpos.st_ctrl.in.b_ausfahren:= TRUE;
		END_IF

		(*-----------------------Weiterschaltbedingungen----------------------------*)
		IF zyl_Indexier_Bestueckpos.st_ctrl.out.b_ausgefahren AND
			zyl_Indexier_Einlauf.st_ctrl.out.b_ausgefahren THEN
			zyl_Indexier_Bestueckpos.st_ctrl.in.b_ausfahren:= FALSE;
			fb_state_entry.i16_next_step := 310;
		END_IF

(*=======================================================*)
	310: fb_state_entry.s_debugtext := 'warten auf Achse bereit';

		(*-----------------------Weiterschaltbedingungen----------------------------*)
		IF	axis_transport_wt_achse.st_ctrl.out.b_bereit AND
			NOT axis_transport_wt_achse.st_ctrl.out.b_busy  AND
			NOT axis_transport_wt_achse.st_ctrl.in.b_start THEN
			fb_state_entry.i16_next_step := 320;
		END_IF

(*=======================================================*)
	320: fb_state_entry.s_debugtext := 'Fahre Achse wieder zurück';

		IF fb_state_entry.E THEN
			ST_WT_Transport_Achse.lr_Achspos_in:=gst_datensatz.st_md.st_md_transport_wt_achse.lr_startposition;
			ST_WT_Transport_Achse.lr_Velo_in:= gst_datensatz.st_md.r_geschwindigkeit_achse_transport;
			ST_WT_Transport_Achse.enu_cmd_in:=MOVE_ABSOLUTE;
			axis_transport_wt_achse.st_ctrl.in.b_start := TRUE;
		END_IF

		(*-----------------------Weiterschaltbedingungen----------------------------*)
		IF	axis_transport_wt_achse.st_ctrl.out.b_busy  THEN
			axis_transport_wt_achse.st_ctrl.in.b_start := FALSE;
			fb_state_entry.i16_next_step := 330;
		END_IF

(*=======================================================*)
	330: fb_state_entry.s_debugtext := 'warten auf Achse hinten fertig';

		(*-----------------------Weiterschaltbedingungen----------------------------*)
		IF	axis_transport_wt_achse.st_ctrl.out.b_fertig  THEN
			fb_state_entry.i16_next_step := BEREIT;
		END_IF

(*=======================================================*)
	500: fb_state_entry.s_debugtext := 'Warte bis angekommen an Stopper';
		IF fb_state_entry.E THEN
			bm_warte_auf_wt_an_stopper := TRUE;
		END_IF

		IF e_wt_im_aktionsfeld AND NOT fb_ton_wz.Q THEN
			fb_ton_wz.PT := t#3s;
			fb_ton_wz.IN := TRUE;
		END_IF

		(*-----------------------Weiterschaltbedingungen----------------------------*)
		IF fb_ton_wt_auf_beladepos.Q THEN
			fb_ton_wz.IN := FALSE;
			fb_state_entry.i16_next_step := 510;
		END_IF

		(*Abfrage auf Sensorfehler des Beladepositionssensors *)
		IF NOT e_wt_im_aktionsfeld  AND fb_ton_wz.Q THEN
			sm_sensorfehler_beladepos := TRUE;
			fb_state_entry.i16_next_step := FEHLER;
		END_IF

(*=======================================================*)
	510: fb_state_entry.s_debugtext := 'WT-Zentrierer ausfahren';

		IF fb_state_entry.E THEN
			zyl_wt_zentrierer_tisch.st_ctrl.in.b_ausfahren := TRUE;
		END_IF

		(*-----------------------Weiterschaltbedingungen----------------------------*)
		IF zyl_wt_zentrierer_tisch.st_ctrl.out.b_ausgefahren  THEN
			zyl_wt_zentrierer_tisch.st_ctrl.in.b_ausfahren := FALSE;
			fb_state_entry.i16_next_step := 520;
		END_IF

(*=======================================================*)
	520:	fb_state_entry.s_debugtext := 'Produktion ohne aktiven WT Transport';

		IF fb_state_entry.E THEN
			axis_z_achse.st_ctrl.in.b_start := TRUE;
		END_IF

		(*-----------------------Weiterschaltbedingungen----------------------------*)
		IF axis_z_achse.st_ctrl.out.b_fertig AND NOT fb_state_entry.E THEN
			axis_z_achse.st_ctrl.in.b_start := FALSE;
			stueckzahlen.st_ctrl.in.b_gutteil_produziert := TRUE;
			IF NOT b_Dauertest_Achsen THEN
				fb_state_entry.i16_next_step := BEREIT;
			ELSE
				(* zum Testen der Achsen nach Tausch, Bestückbild "Becherspucken", WKZ ausgebaut, Vorschubkontrolle abeschaltet,
				Bit muss von Programmierer geforct werden, zum Beenden Schlüsselschalter auf HAND und Zelle neu starten *)
				fb_state_entry.i16_next_step := 500;	(* Dauertest *)
			END_IF
		END_IF

(*=======================================================*)
	FEHLER:
		IF fb_state_entry.E THEN
			st_ctrl_out.b_fehler := TRUE;
			fb_ton_quitt.IN := FALSE;
			zyl_wt_zentrierer_tisch.st_ctrl.in.b_quittieren := FALSE;
			zyl_Indexier_Bestueckpos.st_ctrl.in.b_quittieren := FALSE;
			(*ST_Markiere_WT_NIO();*)
		END_IF

		(*-----------------------Weiterschaltbedingungen----------------------------*)
		IF st_ctrl_in.b_quitt AND NOT fb_state_entry.E THEN
			st_ctrl_out.b_fehler := FALSE;
			zyl_wt_zentrierer_tisch.st_ctrl.in.b_quittieren := TRUE;
			zyl_Indexier_Bestueckpos.st_ctrl.in.b_quittieren := TRUE;
			fb_ton_quitt.IN := TRUE;
		END_IF

		IF fb_ton_quitt.Q THEN
			fb_ton_quitt.IN := FALSE;
			fb_state_entry.i16_next_step := INIT;
		END_IF

(*=======================================================*)
	STOP:
		IF fb_state_entry.E THEN
			fb_ton_quitt.IN := FALSE;
			st_ctrl_out.b_kontroller_start := FALSE;
			zyl_wt_zentrierer_tisch.st_ctrl.in.b_quittieren := FALSE;
			zyl_Indexier_Bestueckpos.st_ctrl.in.b_quittieren := FALSE;

			(*ST_Markiere_WT_NIO();*)
		END_IF

		(*-----------------------Weiterschaltbedingungen----------------------------*)
		IF st_ctrl_in.b_quitt AND NOT fb_state_entry.E THEN
			fb_ton_quitt.IN := TRUE;
			zyl_wt_zentrierer_tisch.st_ctrl.in.b_quittieren := TRUE;
			zyl_Indexier_Bestueckpos.st_ctrl.in.b_quittieren := TRUE;
		END_IF

		IF fb_ton_quitt.Q THEN
			fb_ton_quitt.IN := FALSE;
			fb_state_entry.i16_next_step := INIT;
		END_IF
END_CASE

fb_state_entry(
	i16_next_step:= ,
	i16_pos:= 2,
	s_debugtext:= ,
	E=> ,
	X=> ,
	i16_step=> ,
	i16_last_step=> );

fb_ton_abfrage_wt_auf_beladepos (IN:=bm_abfrage_wt_auf_beladepos,PT:=t#30s);
fb_ton_warte_auf_wt_an_stopper (IN:=bm_warte_auf_wt_an_stopper,PT:=t#30s);

IF st_config.b_config_fertig THEN
	(* Fehlermeldungen ab dem Startindex in das globale Störmeldungsarray schreiben *)
	garr_stoermeldungen[st_config.i16_meld_startindex + 0] := sm_wt_hat_beladepos_nicht_verlassen;
	garr_stoermeldungen[st_config.i16_meld_startindex + 1] := sm_tagnummer_ungueltig;
	garr_stoermeldungen[st_config.i16_meld_startindex + 2] := sm_wt_hat_kein_tag;
	garr_stoermeldungen[st_config.i16_meld_startindex + 3] := FALSE;
	garr_stoermeldungen[st_config.i16_meld_startindex + 4] := sm_tagreader_nicht_fertig;
	garr_stoermeldungen[st_config.i16_meld_startindex + 5] := sm_keine_bandfreigabe;
	garr_stoermeldungen[st_config.i16_meld_startindex + 6] := FALSE;
	garr_stoermeldungen[st_config.i16_meld_startindex + 7] := FALSE;
	garr_stoermeldungen[st_config.i16_meld_startindex + 8] := FALSE;
	garr_stoermeldungen[st_config.i16_meld_startindex + 9] := FALSE;
	garr_stoermeldungen[st_config.i16_meld_startindex + 10] := FALSE;
	garr_stoermeldungen[st_config.i16_meld_startindex + 11] := FALSE;
	garr_stoermeldungen[st_config.i16_meld_startindex + 12] := FALSE;
	garr_stoermeldungen[st_config.i16_meld_startindex + 13] := FALSE;
	garr_stoermeldungen[st_config.i16_meld_startindex + 14] := FALSE;
	garr_stoermeldungen[st_config.i16_meld_startindex + 15] := FALSE;
	garr_stoermeldungen[st_config.i16_meld_startindex + 16] := FALSE;
	garr_stoermeldungen[st_config.i16_meld_startindex + 17] := FALSE;
	garr_stoermeldungen[st_config.i16_meld_startindex + 18] := FALSE;
	garr_stoermeldungen[st_config.i16_meld_startindex + 19] := FALSE;
	
